(*******************************************************************************************************************)
//											Non operational system state
(*******************************************************************************************************************)
IF (gu8_SystemState = STANDBY_SYS OR gu8_SystemState = ERROR_SYS OR gu8_SystemState = OFF_SYS) THEN
	hq_BatteryDischargeMain_Rq			:=	FALSE;
	hq_Battery1ChargePrecharge_Rq		:=	FALSE;
	hq_Battery1ChargeMain_Rq			:=	FALSE;
	hq_Battery2ChargePrecharge_Rq		:=	FALSE;
	hq_BatteryDischargePrecharge_Rq		:=	FALSE;
	hq_Battery2ChargeMain_Rq			:=	FALSE;
	hton_Precharge_Timer				(IN := FALSE, PT := T#0MS);
	hton_PrechargeDisconnectBMS1_Timer	(IN := FALSE, PT := T#0MS);
	hton_PrechargeDisconnectBMS2_Timer	(IN := FALSE, PT := T#0MS);
	hton_Contactor_Delay				(IN := FALSE, PT := T#0MS);
	
(*******************************************************************************************************************)
//												System State Pre-Discharge
(*******************************************************************************************************************)
ELSIF (gu8_SystemState = DRIVE_SYS AND gr_BMS_BatteryVoltage > 0) THEN
	hr_MainConnectionVoltage	:=	gr_BMS_BatteryVoltage * PRECHARGEEND_VOLTAGE_PERC;
	hton_Contactor_Delay						(IN := TRUE, PT := T#500MS);
	IF (hton_Contactor_Delay.Q = TRUE) THEN
		IF ((gr_Sevcon1_DCLink_Voltage <= hr_MainConnectionVoltage OR
			 gr_Sevcon2_DCLink_Voltage <= hr_MainConnectionVoltage OR
			gu16_MCU_HighPowerVoltage <= hr_MainConnectionVoltage) AND
			DO_q_BatteryDischargeMain_DO = FALSE) THEN
			hq_BatteryDischargePrecharge_Rq	:=	TRUE;
			hton_PrechargeDisconnect_Timer		(IN := FALSE, PT := T#0MS);
			hton_MainContactorConnection_Delay	(IN := FALSE, PT := T#0MS);
(*******************************************************************************************************************)
//												System State Discharge
(*******************************************************************************************************************)			
		ELSIF ((gr_Sevcon1_DCLink_Voltage > hr_MainConnectionVoltage AND
				gr_Sevcon2_DCLink_Voltage > hr_MainConnectionVoltage AND
				gu16_MCU_HighPowerVoltage > hr_MainConnectionVoltage) OR
				DO_q_BatteryDischargeMain_DO = TRUE) THEN
			hton_MainContactorConnection_Delay(IN := TRUE, PT := T#100MS);
			IF (hton_MainContactorConnection_Delay.Q = TRUE) THEN
				hq_BatteryDischargeMain_Rq		:=	TRUE;
				hton_PrechargeDisconnect_Timer(IN := TRUE, PT := T#1S);
				IF (hton_PrechargeDisconnect_Timer.Q = TRUE) THEN
					hq_BatteryDischargePrecharge_Rq	:=	FALSE;
				END_IF
			END_IF
		ELSE
			hq_BatteryDischargeMain_Rq		:=	FALSE;
		END_IF
	END_IF
	hq_Battery1ChargePrecharge_Rq			:=	FALSE;
	hq_Battery1ChargeMain_Rq				:=	FALSE;
	hq_Battery2ChargePrecharge_Rq			:=	FALSE;
	hq_Battery2ChargeMain_Rq				:=	FALSE;
(*******************************************************************************************************************)
//												System State Charge
(******************************************************************************************************************)
ELSIF ((gu8_SystemState = PLUGIN_SYS AND
		Brusa1_Rx.S_ACDet = TRUE AND
		Brusa2_Rx.S_ACDet = TRUE AND
		gr_BMS_BatteryVoltage > 0)) THEN// Reset charge sequence if BMS safety drops out
		hton_Contactor_Delay(IN := DO_q_DrivetrainKL15C_DO, PT := T#500MS);
	IF (hton_Contactor_Delay.Q = TRUE) THEN
(*******************************************************************************************************************)
//												System State Pre-Charge Master
(******************************************************************************************************************)	
		IF OrionBMS1_RxConversion.Safety_OK THEN // Check that BMS1 safety is ok
			IF (Brusa1_RxConversion.DCHVVoltAct <= (gr_BMS1_Voltage * PRECHARGEEND_VOLTAGE_PERC) AND
				(DO_q_Battery1ChargeMain_DO = FALSE)) THEN
				hq_Battery1ChargePrecharge_Rq		  := TRUE;
(*******************************************************************************************************************)
//												System State Main-Charge Master
(******************************************************************************************************************)					
			ELSIF (Brusa1_RxConversion.DCHVVoltAct > (gr_BMS1_Voltage * PRECHARGEEND_VOLTAGE_PERC) OR
				DO_q_Battery1ChargeMain_DO) THEN
				hq_Battery1ChargeMain_Rq			  := TRUE;
				hton_PrechargeDisconnectBMS1_Timer(IN := TRUE, PT := T#1S);
				IF (hton_PrechargeDisconnectBMS1_Timer.Q) THEN
						hq_Battery1ChargePrecharge_Rq := FALSE;
				END_IF
			END_IF
		END_IF
(*******************************************************************************************************************)
//												System State Pre-Charge Slave
(******************************************************************************************************************)	
		IF OrionBMS2_RxConversion.Safety_OK THEN // Check that BMS2 safety is ok
			IF (Brusa2_RxConversion.DCHVVoltAct <= (gr_BMS2_Voltage * PRECHARGEEND_VOLTAGE_PERC) AND
				(DO_q_Battery2ChargeMain_DO = FALSE)) THEN
				hq_Battery2ChargePrecharge_Rq		  := TRUE;
(*******************************************************************************************************************)
//												System State Main-Charge Master
(******************************************************************************************************************)					
			ELSIF (Brusa2_RxConversion.DCHVVoltAct > (gr_BMS2_Voltage * PRECHARGEEND_VOLTAGE_PERC) OR
				DO_q_Battery2ChargeMain_DO) THEN
				hq_Battery2ChargeMain_Rq			  := TRUE;	
				hton_PrechargeDisconnectBMS2_Timer(IN := TRUE, PT := T#1S);
				IF (hton_PrechargeDisconnectBMS2_Timer.Q) THEN
					hq_Battery2ChargePrecharge_Rq	  := FALSE;
				END_IF
			END_IF
		END_IF
	ELSE
(*******************************************************************************************************************)
//												System Swich off all Contactor requests
(******************************************************************************************************************)			
		hq_Battery1ChargePrecharge_Rq		:=	FALSE;
		hq_Battery2ChargePrecharge_Rq		:=	FALSE;
		hq_Battery1ChargeMain_Rq			:=	FALSE;
		hq_Battery2ChargeMain_Rq			:=	FALSE;
	END_IF
	hq_BatteryDischargeMain_Rq				:=	FALSE;
	hq_BatteryDischargePrecharge_Rq			:=	FALSE;
ELSE
	hq_BatteryDischargeMain_Rq				:=	FALSE;
	hq_Battery1ChargePrecharge_Rq			:=	FALSE;
	hq_Battery1ChargeMain_Rq				:=	FALSE;
	hq_Battery2ChargePrecharge_Rq			:=	FALSE;
	hq_BatteryDischargePrecharge_Rq			:=	FALSE;
	hq_Battery2ChargeMain_Rq				:=	FALSE;
	hton_Precharge_Timer					(IN := FALSE, PT := T#0MS);
	hton_Contactor_Delay					(IN := FALSE, PT := T#0MS);
END_IF

(*******************************************************************************************************************)
//											Set the actual output values
// 		Current protection so if system current is over a certain value maintain contactor state to prevent welds
(******************************************************************************************************************)	
IF ((DOS_q_BatteryDischargeMain_DO <> hq_BatteryDischargeMain_Rq) AND
	(ABS(gs16_BMS_BatteryCurrent) > CONTACTORSWITCH_CURRENT_LIMIT)) THEN
	DO_q_BatteryDischargeMain_DO	:=	DOS_q_BatteryDischargeMain_DO;
ELSE
	DO_q_BatteryDischargeMain_DO	:=	hq_BatteryDischargeMain_Rq;
END_IF

IF ((DOS_q_Battery1ChargeMain_DO <> hq_Battery1ChargeMain_Rq) AND
	(ABS(gs16_BMS_BatteryCurrent) > CONTACTORSWITCH_CURRENT_LIMIT)) THEN
	DO_q_Battery1ChargeMain_DO	:=	DOS_q_Battery1ChargeMain_DO;
ELSE
	DO_q_Battery1ChargeMain_DO	:=	hq_Battery1ChargeMain_Rq;
END_IF

IF (DOS_q_Battery2ChargeMain_DO <> hq_Battery2ChargeMain_Rq AND
	(ABS(gs16_BMS_BatteryCurrent) > CONTACTORSWITCH_CURRENT_LIMIT)) THEN
	DO_q_Battery2ChargeMain_DO	:=	DOS_q_Battery2ChargeMain_DO;
ELSE
	DO_q_Battery2ChargeMain_DO	:=	hq_Battery2ChargeMain_Rq;
END_IF
(*******************************************************************************************************************)
//						Precharge contactors can change states to allow system connection								
(******************************************************************************************************************)		
DO_q_BatteryDischargePrecharge_DO	:=	hq_BatteryDischargePrecharge_Rq;
DO_q_Battery1ChargePrecharge_DO		:=	hq_Battery1ChargePrecharge_Rq;
DO_q_Battery2ChargePrecharge_DO		:=	hq_Battery2ChargePrecharge_Rq;

END_PROGRAM

// Application/UserCode/Brusa/Brusa2_Comms/Brusa2_RxConversion
PROGRAM Brusa2_RxConversion
VAR
ACVoltL1Act		:	UINT;
	ACVoltL2Act		:	UINT;
	ACVoltL3Act		:	UINT;
	ACCurrL1Act		:	SINT;
	ACCurrL2Act		:	SINT;
	ACCurrL3Act		:	SINT;
	ACPowTotAct		:	UINT;
	MaxTempAct		:	INT;
	TempCon			:	INT;
	DCHVAhAct			:	REAL;
	DCHVVoltAct			:	REAL;
	DCHVCurrAct			:	REAL;
	ACCurrMaxAct		:	REAL;
	ACCurrHWAvl			:	REAL;
	ACCurrMaxCP			:	REAL;
	TempCoolPlate		:	INT;		
END_VAR

ACVoltL1Act	:=	USINT_TO_UINT(Brusa2_Rx.ACVoltL1Act_Rx) * 2;
ACVoltL2Act	:=	USINT_TO_UINT(Brusa2_Rx.ACVoltL2Act_Rx) * 2;
ACVoltL3Act	:=	USINT_TO_UINT(Brusa2_Rx.ACVoltL3Act_Rx) * 2;
ACCurrL1Act	:=	USINT_TO_SINT(Brusa2_Rx.ACCurrL1Act_Rx) - 127;
ACCurrL2Act	:=	USINT_TO_SINT(Brusa2_Rx.ACCurrL2Act_Rx) - 127;
ACCurrL3Act	:=	USINT_TO_SINT(Brusa2_Rx.ACCurrL3Act_Rx) - 127;
ACPowTotAct	:=	USINT_TO_UINT(Brusa2_Rx.ACPowTotAct_Rx) * 100;
MaxTempAct	:=	USINT_TO_INT(Brusa2_Rx.MaxTempAct_Rx) - 50;
TempCon		:=	USINT_TO_INT(Brusa2_Rx.TempCon_Rx) - 50;
DCHVAhAct		:=	UINT_TO_REAL(Brusa2_Rx.DCHVAhAct_Rx) * 0.01;
DCHVVoltAct		:=	UINT_TO_REAL(Brusa2_Rx.DCHVVoltAct_Rx) * 0.1;
DCHVCurrAct		:=	UINT_TO_REAL(Brusa2_Rx.DCHVCurrAct_Rx) * 0.1 - 100;
ACCurrMaxAct	:=	UINT_TO_REAL(Brusa2_Rx.ACCurrMaxAct_Rx) * 0.1 -100;
ACCurrHWAvl		:=	USINT_TO_REAL(Brusa2_Rx.ACCurrHWAvl_Rx) * 0.5;
ACCurrMaxCP		:=	UINT_TO_REAL(Brusa2_Rx.ACCurrMaxCP_Rx) * 0.1;
TempCoolPlate	:=	USINT_TO_INT(Brusa2_Rx.TempCoolPlate_Rx) - 50;

END_PROGRAM

// Application/UserCode/Cooling Fan/Fan_Cooling
PROGRAM Fan_Cooling
VAR
	Cooling_Fan_MCU_SP				:	REAL	:=	30; // 30% requested
	Cooling_Fan_BRUSA_Charge_SP		:	REAL	:=	82;
	Cooling_Fan_BellP_Charge_SP		:	REAL	:=	82;	//	BellPower Charger 
	Cooling_Fan_DCDC_SP				:	REAL	:=	45; // Actual C Temp.
	Cooling_Fan_Request				:	BOOL	:=	FALSE;
	Cooling_Fan_DLY_Off				:	TOF;
	Run_On_Time						:	TIME	:=	T#60S;
END_VAR

(*****************************************************************************************************************)
//                       				   Radiator Cooling Fan
(*****************************************************************************************************************)

IF		((SUPPLY_Power1/100) > 25.0) AND	(NOT gq_EStop)				AND		// Do not run Fan if battery voltage is Low or EStopped
		(gr_MCU_ThermalIndicator		> Cooling_Fan_MCU_SP)			OR		// MCU
		(Brusa1_RxConversion.MaxTempAct	> Cooling_Fan_BRUSA_Charge_SP) 	OR		// BRUSA 1
		(Brusa2_RxConversion.MaxTempAct > Cooling_Fan_BRUSA_Charge_SP) 	OR		// BRUSA 2
	//	(BellPower_Charging				> Cooling_Fan_BellP_Charge_SP	OR		//	BellPower Charging	
		(BELDCDC_RxConversion.TempCoolant	> Cooling_Fan_DCDC_SP)		OR		// DCDC	
		HMI_Rx.PB_Cooling_Fan_Request									THEN	// Request from HMI
	
		Cooling_Fan_Request				:= TRUE;								// Fan Requested
ELSE
		Cooling_Fan_Request 			:= FALSE;								// Fan not Required
END_IF

		Cooling_Fan_DLY_Off		(IN := Cooling_Fan_Request, PT :=Run_On_Time);	// Fan run on time   (****provides hysteresis***)
IF 		(Cooling_Fan_DLY_Off.Q = TRUE) 									THEN
		DO_q_DrivetrainCoolingFan_DO	:=	TRUE;								// Fan Relay On
ELSE 
		DO_q_DrivetrainCoolingFan_DO	:=	FALSE;								// Fan Relay Off
END_IF

END_PROGRAM

// Application/UserCode/Cruise Control/CruiseControl
PROGRAM CruiseControl
VAR
	Cruise_Control_Button_DI: BOOL := FALSE;
	RS_CC: RS;
	CC_SetSpeed: REAL := 0;
	CC_Active: BOOL := FALSE;
	CC_VehicleSpeed: REAL := 0;
	SR_CC: SR;
	F_TRIG_CC_Set: F_TRIG;
	R_TRIG_CC_Set: R_TRIG;
	TESTSpeed: REAL := 0;
END_VAR

//Cruise Control

F_TRIG_CC_Set (CLK := DI_q_PB_Cruise_Control_DI);
R_TRIG_CC_Set (CLK := DI_q_PB_Cruise_Control_DI);

IF R_TRIG_CC_Set.Q AND gq_BrakeSwitch = FALSE AND (gu8_RegenSelector < 1) AND gu8_TractionLoss = 0 AND gu8_StabilityLoss = 0 THEN //LM added stab and trac event to cancel
	CC_Active := TRUE;
ELSIF CC_Active = TRUE THEN
	IF gq_BrakeSwitch = TRUE OR gu8_RegenSelector > 0 OR gu8_TractionLoss = 1 OR gu8_StabilityLoss = 1 THEN
	CC_Active := FALSE;
	END_IF
END_IF

IF CC_Active = TRUE THEN
	RS_CC (SET := DI_q_PB_Cruise_Control_DI = TRUE, RESET1 := F_TRIG_CC_Set.Q = TRUE);
END_IF

IF R_TRIG_CC_Set.Q = TRUE THEN
	SR_CC (SET1 := R_TRIG_CC_Set.Q = TRUE, RESET := (gq_BrakeSwitch = TRUE AND gu8_RegenSelector = 1));
END_IF

//IF SR_CC.Q1 = TRUE THEN
//	CC_SetSpeed := TESTSpeed;//gr_VehicleSpeed_kmph;
//END_IF

IF RS_CC.Q1 = TRUE THEN
	CC_SetSpeed := LIMIT (5, gr_VehicleSpeed_kmph, 57);//TESTSpeed;
END_IF

END_PROGRAM

// Application/UserCode/ePTO/ePTO_Control_1
PROGRAM ePTO_Control_1
VAR
	hu16_TORQUEREFHIGH	: UINT	:=	90; (*%*)
	hu16_TORQUEREFLOW	: UINT	:=	0;	(*%*)
	hu16_SPEEDTARGET	: UINT	:=	1150; (*RPM*)
	hs16_FAN_On_Temp	: INT	:=	60; (*degC*)
	hs16_FAN_Off_Temp	: INT	:=	50;	(*degC*)
	
	hton_CANOpen_Start_Timer	:	TON;
	hton_CANOpen_StartCommand_OtherAddress_Timer	:	TON;
	hu16_IdleSpeedTarget: UINT := 250;
	BinLiftTimer: TON;
	BinLiftTime: TIME := t#3s;
END_VAR


gu16_TrqHi	:=	(hu16_TORQUEREFHIGH * 50) + 5000;
gu16_TrqLo	:=	(hu16_TORQUEREFLOW * 50) + 5000;
gu8_Asym_Limits	:=	16#20;

IF ((gs16_InverterTemp > hs16_FAN_On_Temp) OR (gs16_MotorTemp > hs16_FAN_On_Temp)) THEN
	gu8_DIGITAL1	:=	16#80;
ELSIF ((gs16_InverterTemp < hs16_FAN_Off_Temp) AND (gs16_MotorTemp < hs16_FAN_Off_Temp)) THEN
	gu8_DIGITAL1	:=	16#0;
END_IF

BinLiftTimer (IN:= (gq_Gear_Drive = TRUE OR gq_Gear_Reverse = TRUE), PT:= BinLiftTime);

IF (DOS_q_BatteryDischargeMain_DO = TRUE) THEN
	(*Activate Motor*)
	IF (gu8_ePTO_ActivationByte <> 0) OR (BinLiftTimer.Q = FALSE AND gq_Gear_Neutral = FALSE) THEN
		gu16_Skai_SpeedTarget	:=	hu16_SPEEDTARGET + 32768;
		gq_ePTO_Activate	:=	TRUE;
	ELSE
		gu16_Skai_SpeedTarget	:=	hu16_IdleSpeedTarget + 32768; (*added to allow permanent running of ePTO*)
		gq_ePTO_Activate	:=	TRUE(*FALSE*);
	END_IF
ELSE
	gu16_Skai_SpeedTarget	:=	32768; (*Offset so value is actually 0*)
	gq_ePTO_Activate	:=	FALSE;
END_IF


(*CANOpen*)
hton_CANOpen_Start_Timer(IN := TRUE, PT := T#5S);
hton_CANOpen_StartCommand_OtherAddress_Timer(IN := hton_CANOpen_Start_Timer.Q, PT := T#1S);
IF (hton_CANOpen_Start_Timer.Q = TRUE) THEN
	gu8_CANOpen_Command	:=	16#01;
	gu8_CANOpen_NodeAddress	:=	16#7A;
ELSIF (hton_CANOpen_StartCommand_OtherAddress_Timer.Q = TRUE) THEN
	gu8_CANOpen_Command	:=	16#01;
	gu8_CANOpen_NodeAddress	:=	16#7B;
ELSE
	gu8_CANOpen_Command	:=	16#81;
	gu8_CANOpen_NodeAddress	:=	16#7A;
END_IF

DO_q_ePTO_Fan_DO	:=	gq_ePTO_Activate;

END_PROGRAM

// Application/UserCode/ePTO/EPTO_Rx_1
PROGRAM EPTO_Rx_1
VAR
	ePTO_Rx			:	Receive_CAN4_STD;
	ePTO_Dennis_Rx	:	Receive_CAN4_EXD;
	SkaiUnit_Temp_Rx	:	Receive_CAN4_STD;
END_VAR


ePTO_Rx		(u32_COBID	:=	16#141,
						q_NewData => ,
						au8_Data => ,
						u8_Length => 		);
						
ePTO_Dennis_Rx (u32_COBID	:=	16#2CFF1355,
						q_NewData => ,
						au8_Data => ,
						u8_Length => 		);
						
SkaiUnit_Temp_Rx (u32_COBID	:=	16#1BA,
						q_NewData => ,
						au8_Data => ,
						u8_Length => 		);

IF (gu8_ChassisType = CHASSIS_DENNIS) THEN
	gu8_ePTO_ActivationByte	:=	ePTO_Dennis_Rx.au8_Data[3]; (*4*)
ELSE
	gu8_ePTO_ActivationByte	:=	ePTO_Rx.au8_Data[4];				
END_IF					

gs16_InverterTemp	:= SkaiUnit_Temp_Rx.au8_Data[0] - 40;
gs16_MotorTemp		:= SkaiUnit_Temp_Rx.au8_Data[1] - 40; (*Use this for the ePTO activation instead of the boolean trigger*)

END_PROGRAM

// Application/UserCode/ePTO/EPTO_Tx_1
PROGRAM EPTO_Tx_1
VAR
	MercCurrentGear1_Tx	:	EPEC_CANVXD.Msg;
	MercLHFWheelSpd_Tx	:	EPEC_CANVXD.Msg;
	MercCurrentGear2_Tx	:	EPEC_CANVXD.Msg;
	MercControlRPM_Tx	:	EPEC_CANVXD.Msg;
	ePTO_OilRq_Tx		:	EPEC_CANVXD.Msg;
	ePTO_Speed_47A_Tx	:	EPEC_CANVXD.Msg;
	ePTO_Torque_57A_Tx	:	EPEC_CANVXD.Msg;
	ePTO_NMT_Tx			:	EPEC_CANVXD.Msg;
	
	
	hton_MercePTO_TxTimer	:	TON;
END_VAR


{region "Data Allocation"}
(*Merc*)
MercCurrentGear1_Tx.ID := 16#18FE61EB OR EPEC_CANVXD.MASK_29BIT;
MercCurrentGear1_Tx.Data[0]	:=	0;
MercCurrentGear1_Tx.Data[1]	:=	gu8_CurrentGear2;
MercCurrentGear1_Tx.Data[2]	:=	0;
MercCurrentGear1_Tx.Data[3]	:=	0;
MercCurrentGear1_Tx.Data[4]	:=	0;
MercCurrentGear1_Tx.Data[5]	:=	0;
MercCurrentGear1_Tx.Data[6]	:=	0;
MercCurrentGear1_Tx.Data[7]	:=	0;
MercCurrentGear1_Tx.Len		:=	8;

MercLHFWheelSpd_Tx.ID := 16#0CFE5FEB OR EPEC_CANVXD.MASK_29BIT;
MercLHFWheelSpd_Tx.Data[0]	:=	0;
MercLHFWheelSpd_Tx.Data[1]	:=	0;
MercLHFWheelSpd_Tx.Data[2]	:=	0;
MercLHFWheelSpd_Tx.Data[3]	:=	03;
MercLHFWheelSpd_Tx.Data[4]	:=	20;
MercLHFWheelSpd_Tx.Data[5]	:=	0;
MercLHFWheelSpd_Tx.Data[6]	:=	UINT_TO_USINT(gu16_Bob_LeftFront_CAN);
MercLHFWheelSpd_Tx.Data[7]	:=	UINT_TO_USINT(SHR(gu16_Bob_LeftFront_CAN, 8));
MercLHFWheelSpd_Tx.Len		:=	8;

MercCurrentGear2_Tx.ID := 16#14FE80EB OR EPEC_CANVXD.MASK_29BIT;
MercCurrentGear2_Tx.Data[0]	:=	0;
MercCurrentGear2_Tx.Data[1]	:=	gu8_CurrentGear2;
MercCurrentGear2_Tx.Data[2]	:=	0;
MercCurrentGear2_Tx.Data[3]	:=	0;
MercCurrentGear2_Tx.Data[4]	:=	0;
MercCurrentGear2_Tx.Data[5]	:=	0;
MercCurrentGear2_Tx.Data[6]	:=	0;
MercCurrentGear2_Tx.Data[7]	:=	0;
MercCurrentGear2_Tx.Len		:=	8;

MercControlRPM_Tx.ID := 16#0CFE62C9 OR EPEC_CANVXD.MASK_29BIT;
MercControlRPM_Tx.Data[0]	:=	0;
MercControlRPM_Tx.Data[1]	:=	0;
MercControlRPM_Tx.Data[2]	:=	0;
MercControlRPM_Tx.Data[3]	:=	16#FA;
MercControlRPM_Tx.Data[4]	:=	0;
MercControlRPM_Tx.Data[5]	:=	0;
MercControlRPM_Tx.Data[6]	:=	0;
MercControlRPM_Tx.Data[7]	:=	0;
MercControlRPM_Tx.Len		:=	8;
	 
ePTO_OilRq_Tx.ID			:=	16#0CFF1355 OR EPEC_CANVXD.MASK_29BIT;
ePTO_OilRq_Tx.Data[0]		:=	0;
ePTO_OilRq_Tx.Data[1]		:=	0;
ePTO_OilRq_Tx.Data[2]		:=	0;
ePTO_OilRq_Tx.Data[3]		:=	0;
ePTO_OilRq_Tx.Data[3].0		:=	gq_ePTO_Activate;
ePTO_OilRq_Tx.Data[4]		:=	0;
ePTO_OilRq_Tx.Data[5]		:=	0;
ePTO_OilRq_Tx.Data[6]		:=	0;
ePTO_OilRq_Tx.Data[7]		:=	0;
ePTO_OilRq_Tx.Len			:=	8;
(**)


ePTO_Speed_47A_Tx.ID		:=	16#47A;
ePTO_Speed_47A_Tx.Data[0]	:=	UINT_TO_USINT(gu16_TrqHi);
ePTO_Speed_47A_Tx.Data[1]	:=	UINT_TO_USINT(SHR(gu16_TrqHi, 8));
ePTO_Speed_47A_Tx.Data[2]	:=	UINT_TO_USINT(gu16_Skai_SpeedTarget);
ePTO_Speed_47A_Tx.Data[3]	:=	UINT_TO_USINT(SHR(gu16_Skai_SpeedTarget, 8));
ePTO_Speed_47A_Tx.Data[4]	:=	(BOOL_TO_USINT(gq_ePTO_Activate) * 2);
ePTO_Speed_47A_Tx.Data[5]	:=	gu8_Asym_Limits + gu8_DIGITAL1;
ePTO_Speed_47A_Tx.Data[6]	:=	0;
ePTO_Speed_47A_Tx.Data[7]	:=	0;
ePTO_Speed_47A_Tx.Len		:=	8;
	 
ePTO_Torque_57A_Tx.ID		:=	16#57A;
ePTO_Torque_57A_Tx.Data[0]	:=	UINT_TO_USINT(gu16_TrqHi);
ePTO_Torque_57A_Tx.Data[1]	:=	UINT_TO_USINT(SHR(gu16_TrqHi, 8));
ePTO_Torque_57A_Tx.Data[2]	:=	UINT_TO_USINT(gu16_TrqLo);
ePTO_Torque_57A_Tx.Data[3]	:=	UINT_TO_USINT(SHR(gu16_TrqLo, 8));
ePTO_Torque_57A_Tx.Data[4]	:=	0;
ePTO_Torque_57A_Tx.Data[5]	:=	0;
ePTO_Torque_57A_Tx.Data[6]	:=	0;
ePTO_Torque_57A_Tx.Data[7]	:=	0;
ePTO_Torque_57A_Tx.Len		:=	8;

(*CANOpen*)
ePTO_NMT_Tx.ID				:=	16#00;
ePTO_NMT_Tx.Data[0]			:=	gu8_CANOpen_Command;
ePTO_NMT_Tx.Data[1]			:=	gu8_CANOpen_NodeAddress;
ePTO_NMT_Tx.Len				:=	8;
{endregion}

	 
(**************************************************************************************************************************************************)
{region "Send Messages"}
(*Transmit*)
hton_MercePTO_TxTimer(IN := NOT(hton_MercePTO_TxTimer.Q), PT := T#100MS);
IF (hton_MercePTO_TxTimer.Q = TRUE) THEN
	IF (gu8_ChassisType = CHASSIS_BOB OR gu8_ChassisType = CHASSIS_ESTARGLIDER) THEN
		G_CAN4_Channel.SendMessage(i_pMSG:=ADR(MercCurrentGear1_Tx)); 
		G_CAN4_Channel.SendMessage(i_pMSG:=ADR(MercLHFWheelSpd_Tx)); 
		G_CAN4_Channel.SendMessage(i_pMSG:=ADR(MercCurrentGear2_Tx)); 
		G_CAN4_Channel.SendMessage(i_pMSG:=ADR(MercControlRPM_Tx));
	ELSIF (gu8_ChassisType = CHASSIS_DENNIS) THEN
		;
	END_IF
 
	G_CAN4_Channel.SendMessage(i_pMSG:=ADR(ePTO_Speed_47A_Tx));
	G_CAN4_Channel.SendMessage(i_pMSG:=ADR(ePTO_Torque_57A_Tx)); 
	G_CAN4_Channel.SendMessage(i_pMSG:=ADR(ePTO_OilRq_Tx)); 
		 
	G_CAN4_Channel.SendMessage(i_pMSG:=ADR(ePTO_NMT_Tx)); 
END_IF

{end_region}

END_PROGRAM

// Application/UserCode/Fault Handler/FaultDetection_1
PROGRAM FaultDetection_1
VAR
	hq_Dennis_CommsErr			:	BOOL;
	gq_BMS1_Orion_Error			:	BOOL;
	gq_BMS2_Orion_Error			:	BOOL;
	gq_BMS1_Error				:	BOOL;
	gq_BMS2_Error				:	BOOL;
	gq_BMS_Error				:	BOOL;
	gq_DCDC_Bel_Error			:	BOOL;
	gq_MCU_Error				:	BOOL;
	gq_NLG1_Error				:	BOOL;
	gq_NLG2_Error				:	BOOL;
	gq_Sevcon_Steer_Error		:	BOOL;
	gq_Sevcon_Compressor_Error	:	BOOL;
	gq_LV_Error					:	BOOL;// 24V Batteries too Low Error
END_VAR
VAR CONSTANT
	FAULTOFF_STAT				:	USINT	:=	13;
	Low_24V_Battery_Voltage_SP	:	USINT	:=	21;
END_VAR

(**********************************************************************************)
//									Faults & Errors
(**********************************************************************************)

(**********************************************************************************)
// 									Orion BMS1 Faults
(**********************************************************************************)

IF (gu8_BMSType = BMS_ORION) THEN
	IF(	//OrionBMS1_DTCFlag1_0A07_DischargeLimitEnforcementFault= TRUE OR
		OrionBMS1_DTCFlag1_0A08_ChargerSafetyRelayFault			= TRUE OR
		OrionBMS1_DTCFlag1_0A09_InternalHardwareFault			= TRUE OR
		OrionBMS1_DTCFlag1_0A0A_InternalHeatskinkThermistorFault= TRUE OR
		OrionBMS1_DTCFlag1_0A0B_InternalSoftwareFault			= TRUE OR
		OrionBMS1_DTCFlag1_0A0C_HighestCellVoltageTooHighFault	= TRUE OR 
		OrionBMS1_DTCFlag1_0A0E_LowestCellVoltageTooLowFault	= TRUE OR	
		OrionBMS1_DTCFlag1_0A10_PackTooHotFault					= TRUE OR	
		(*DTC2 Flags*)
		OrionBMS1_DTCFlags2_0A1F_InternalCommunicationFault		= TRUE OR	
		//OrionBMS1_DTCFlags2_0A12_CellBalancingStruckOffFault	= TRUE OR	
		//OrionBMS1_DTCFlags2_0A80_WeakCellFault				= TRUE OR*)
		OrionBMS1_DTCFlags2_0AFA_LowCellVoltageFault			= TRUE OR			
		OrionBMS1_DTCFlags2_0A04_OpenWiringFault				= TRUE OR
		OrionBMS1_DTCFlags2_0AC0_CurrentSensorFault				= TRUE OR				
		OrionBMS1_DTCFlags2_0A0D_HighestCellVoltageOver5vFault	= TRUE OR		
		OrionBMS1_DTCFlags2_0A0F_CellASICFault					= TRUE OR
		OrionBMS1_DTCFlags2_0A02_WeakPackFault					= TRUE OR				
		//OrionBMS1_DTCFlags2_0A81_FanMonitorFault				= TRUE OR				
		//OrionBMS1_DTCFlags2_0A9C_ThermistorFault				= TRUE OR			
		OrionBMS1_DTCFlags2_0100_ExternalCommunicationFault		= TRUE OR		
		OrionBMS1_DTCFlags2_0560_RedundantPowerSupplyFault		= TRUE OR	
		OrionBMS1_DTCFlags2_0AA6_HighVoltageIsolatonFault		= TRUE OR
		OrionBMS1_DTCFlags2_0A05_InputPowerSupplyFault			= TRUE OR	
		//OrionBMS1_DTCFlags2_0A06_ChargeLimitEnforcementFault	= TRUE OR
		gq_OrionBMS1_CommsLoss 									= TRUE) THEN
			gq_BMS1_Orion_Error									:=	TRUE;
	ELSE
			gq_BMS1_Orion_Error									:=	FALSE;
	END_IF

(**********************************************************************************)	
// 									Orion BMS2 Faults	
(**********************************************************************************)

	IF(//OrionBMS2_DTCFlag1_0A07_DischargeLimitEnforcementFault= TRUE OR
		OrionBMS2_DTCFlag1_0A08_ChargerSafetyRelayFault			= TRUE OR
		OrionBMS2_DTCFlag1_0A09_InternalHardwareFault			= TRUE OR
		OrionBMS2_DTCFlag1_0A0A_InternalHeatskinkThermistorFault= TRUE OR
		OrionBMS2_DTCFlag1_0A0B_InternalSoftwareFault			= TRUE OR
		OrionBMS2_DTCFlag1_0A0C_HighestCellVoltageTooHighFault	= TRUE OR 
		OrionBMS2_DTCFlag1_0A0E_LowestCellVoltageTooLowFault	= TRUE OR	
		OrionBMS2_DTCFlag1_0A10_PackTooHotFault					= TRUE OR	
		(*DTC2 Flags*)
		OrionBMS2_DTCFlags2_0A1F_InternalCommunicationFault		= TRUE OR	
		//OrionBMS2_DTCFlags2_0A12_CellBalancingStruckOffFault	= TRUE OR	
		//OrionBMS2_DTCFlags2_0A80_WeakCellFault				= TRUE OR
		OrionBMS2_DTCFlags2_0AFA_LowCellVoltageFault			= TRUE OR			
		OrionBMS2_DTCFlags2_0A04_OpenWiringFault				= TRUE OR
		OrionBMS2_DTCFlags2_0AC0_CurrentSensorFault				= TRUE OR				
		OrionBMS2_DTCFlags2_0A0D_HighestCellVoltageOver5vFault	= TRUE OR		
		OrionBMS2_DTCFlags2_0A0F_CellASICFault					= TRUE OR
		OrionBMS2_DTCFlags2_0A02_WeakPackFault					= TRUE OR				
		//OrionBMS2_DTCFlags2_0A81_FanMonitorFault				= TRUE OR				
		//OrionBMS2_DTCFlags2_0A9C_ThermistorFault				= TRUE OR			
		OrionBMS2_DTCFlags2_0100_ExternalCommunicationFault		= TRUE OR		
		OrionBMS2_DTCFlags2_0560_RedundantPowerSupplyFault		= TRUE OR	
		OrionBMS2_DTCFlags2_0AA6_HighVoltageIsolatonFault		= TRUE OR
		OrionBMS2_DTCFlags2_0A05_InputPowerSupplyFault			= TRUE OR	
		//OrionBMS2_DTCFlags2_0A06_ChargeLimitEnforcementFault	= TRUE OR
		gq_OrionBMS2_CommsLoss 									= TRUE) THEN
			gq_BMS2_Orion_Error									:=	TRUE;
	ELSE
			gq_BMS2_Orion_Error									:=	FALSE;
	END_IF
END_IF

(**********************************************************************************)
// 									Orion BMS Faults
(**********************************************************************************)
	 
IF (gq_BMS1_Orion_Error = TRUE) THEN
	gq_BMS1_Error	:=	TRUE;
ELSE
	gq_BMS1_Error	:=	FALSE;		 
END_IF

IF (gq_BMS2_Orion_Error = TRUE) THEN
	gq_BMS2_Error	:=	TRUE;
ELSE 
	gq_BMS2_Error	:=	FALSE;
END_IF

IF (gq_BMS1_Error = TRUE OR gq_BMS2_Error = TRUE) THEN
	gq_BMS_Error	:=	TRUE;
ELSE
	gq_BMS_Error	:=	FALSE;
END_IF

(**********************************************************************************)
// 									BelPower DCDC Faults
(**********************************************************************************)

IF (BELDCDC_Rx.Fault_InputUV 					= TRUE OR
	BELDCDC_Rx.Fault_InputOV 					= TRUE OR
	(*BELDCDC_Rx.gq_BelDCDC_flt_OutputUV		= TRUE OR*)
	BELDCDC_Rx.Fault_OutputOV 					= TRUE OR
	(*BELDCDC_Rx.gq_BelDCDC_flt_OutputOC 		= TRUE OR*) (*Need to reenable this when possible*)
	BELDCDC_Rx.Fault_OTP 						= TRUE OR
	BELDCDC_Rx.Fault_I2CFault 					= TRUE OR
	BELDCDC_Rx.Fault_CANFault 					= TRUE OR
	BELDCDC_Rx.Fault_EEPROM_CRCFault 			= TRUE OR
	BELDCDC_Rx.Fault_ShortCircuit 				= TRUE OR
	BELDCDC_Rx.Fault_ThermistorFault 			= TRUE OR
	BELDCDC_Rx.Fault_Overload 					= TRUE OR
	BELDCDC_Rx.Fault_OutputOVLatch 				= TRUE OR
	BELDCDC_Rx.Fault_ReversePolarity 			= TRUE OR
	BELDCDC_Rx.Warning_CoolantOTP 				= TRUE OR
	BELDCDC_Rx.Warning_CurrentLimiting 			= TRUE OR
	BELDCDC_Rx.CommsLoss)							THEN
	gq_DCDC_Bel_Error							:=	TRUE;
ELSE
	gq_DCDC_Bel_Error							:=	FALSE;
END_IF

(**********************************************************************************)
// 									MCU  Faults
(**********************************************************************************)

IF (gq_MCU_Fault_PhaseToChassis 		= TRUE OR
	gq_MCU_Fault_InterlockBatteryCable 	= TRUE OR
	gq_MCU_Fault_InterlockMotorCable 	= TRUE OR
	gq_MCU_Fault_DriveCoverWasOpened 	= TRUE OR
	gq_MCU_Fault_PhaseToChassisStatus 	= TRUE OR
	(gq_MCU_CommsLoss = TRUE AND gu8_SystemState = DRIVE_SYS)) THEN
	gq_MCU_Error	:=	TRUE;
ELSE
	gq_MCU_Error	:=	FALSE;
END_IF

(**********************************************************************************)
// 									BRUSA1 Faults
(**********************************************************************************)

IF (gu8_ChargerType = CHARGER_BRUSA) THEN
	IF (Brusa1_Rx.E_WrongHW 		= TRUE OR
		Brusa1_Rx.E_WrongFPGA 		= TRUE OR
		Brusa1_Rx.E_EPGAInit 		= TRUE OR
		Brusa1_Rx.E_NVSRam 			= TRUE OR
		Brusa1_Rx.E_Flash 			= TRUE OR
		Brusa1_Rx.E_OSTrap 			= TRUE OR
		Brusa1_Rx.E_HVIsoPos 		= TRUE OR
		Brusa1_Rx.E_HVIsoNeg 		= TRUE OR
		Brusa1_Rx.E_Internal 		= TRUE OR
		Brusa1_Rx.E_TempInt 		= TRUE OR
		Brusa1_Rx.E_DCHVVoltRed 	= TRUE OR
		Brusa1_Rx.E_IntSupply 		= TRUE OR
		Brusa1_Rx.E_CANMsgLost 		= TRUE OR
		Brusa1_Rx.E_CANValue 		= TRUE OR
		Brusa1_Rx.E_ACInterruption 	= TRUE OR
		Brusa1_Rx.E_DCHVVoltRange 	= TRUE OR
		Brusa1_Rx.E_TempCon 		= TRUE OR
		Brusa1_Rx.E_ConLocked 		= TRUE OR
		Brusa1_Rx.E_Interlock 		= TRUE OR
		Brusa1_Rx.E_Crash 			= TRUE OR
		Brusa1_Rx.E_PRELOAD 		= TRUE OR
		Brusa1_Rx.E_BURST 			= TRUE OR
		Brusa1_Rx.E_TPON 			= TRUE OR
		Brusa1_Rx.E_UZK 			= TRUE OR
		Brusa1_Rx.E_LatchFPGA 		= TRUE OR
		Brusa1_Rx.E_OverTemp 		= TRUE OR
		Brusa1_Rx.CommsLoss = TRUE)	 THEN
		gq_NLG1_Error	:=	TRUE;
	ELSE
		gq_NLG1_Error	:=	FALSE;
	END_IF

(**********************************************************************************)	
// 									BRUSA2 Faults
(**********************************************************************************)
			  
	IF (Brusa2_Rx.E_WrongHW 		= TRUE OR
		Brusa2_Rx.E_WrongFPGA 		= TRUE OR
		Brusa2_Rx.E_EPGAInit		= TRUE OR
		Brusa2_Rx.E_NVSRam 			= TRUE OR
		Brusa2_Rx.E_Flash 			= TRUE OR
		Brusa2_Rx.E_OSTrap 			= TRUE OR
		Brusa2_Rx.E_HVIsoPos 		= TRUE OR
		Brusa2_Rx.E_HVIsoNeg 		= TRUE OR
		Brusa2_Rx.E_Internal		= TRUE OR
		Brusa2_Rx.E_TempInt 		= TRUE OR
		Brusa2_Rx.E_DCHVVoltRed 	= TRUE OR
		Brusa2_Rx.E_IntSupply		= TRUE OR
		Brusa2_Rx.E_CANMsgLost		= TRUE OR
		Brusa2_Rx.E_CANValue		= TRUE OR
		Brusa2_Rx.E_ACInterruption = TRUE OR
		Brusa2_Rx.E_DCHVVoltRange 	= TRUE OR
		Brusa2_Rx.E_TempCon			= TRUE OR
		Brusa2_Rx.E_ConLocked 		= TRUE OR
		Brusa2_Rx.E_Interlock 		= TRUE OR
		Brusa2_Rx.E_Crash 			= TRUE OR
		Brusa2_Rx.E_PRELOAD 		= TRUE OR
		Brusa2_Rx.E_BURST 			= TRUE OR
		Brusa2_Rx.E_TPON 			= TRUE OR
	    Brusa2_Rx.E_UZK 			= TRUE OR
		Brusa2_Rx.E_LatchFPGA 		= TRUE OR
		Brusa2_Rx.E_OverTemp 		= TRUE OR
		Brusa2_Rx.CommsLoss 		= TRUE) THEN
		gq_NLG2_Error				:=	TRUE;
	ELSE
			gq_NLG2_Error			:=	FALSE;
	END_IF 
	
END_IF

(**********************************************************************************)
// 									Sevcon Faults
(**********************************************************************************)

IF (gu8_Sevcon1_InverterStatus = FAULTOFF_STAT OR
	(gq_Sevcon1_CommsLoss = TRUE AND gu8_SystemState = DRIVE_SYS)) THEN
	gq_Sevcon_Steer_Error	:=	TRUE;
ELSE
	gq_Sevcon_Steer_Error	:=	FALSE;
END_IF

IF (gu8_Sevcon2_InverterStatus = FAULTOFF_STAT OR
	(gq_Sevcon2_CommsLoss = TRUE AND gu8_SystemState = DRIVE_SYS)) THEN
	gq_Sevcon_Compressor_Error	:=	TRUE;
ELSE
	gq_Sevcon_Compressor_Error	:=	FALSE;
END_IF

(**********************************************************************************)
// 									24VDC Faults
(**********************************************************************************)

IF ((SUPPLY_Power1/100) < Low_24V_Battery_Voltage_SP)  THEN (*SUPPLY_Power1*)
	gq_LV_Error	:=	TRUE;
ELSE
	gq_LV_Error	:=	FALSE; 
END_IF

(**********************************************************************************)
// 									eCompact Faults
(**********************************************************************************)

 IF ((gq_Dennis_CAN1_CommsLoss = TRUE OR CAN4_Rx.Handbrake_Rx_Timer.Q = TRUE) AND
	  gu8_ChassisType = CHASSIS_DENNIS AND gu8_SystemState = DRIVE_SYS) THEN
	hq_Dennis_CommsErr	:=	TRUE;
 ELSE
	hq_Dennis_CommsErr	:=	FALSE;	  
 END_IF

 (**********************************************************************************)
 // 									Global Faults
(**********************************************************************************)
	 
IF (gq_BMS_Error				OR
	gq_DCDC_Bel_Error			OR
	gq_MCU_Error				OR
	Brusa1_Rx.S_Err				OR					//***************************************WRONG!!!!!!!!!!!!!!!!!!!!!!!!!!!
	gq_NLG2_Error				OR
	gq_Sevcon_Steer_Error		OR
	gq_Sevcon_Compressor_Error	OR
	gq_LV_Error					OR
	hq_Dennis_CommsErr			OR
	gq_EStop)	 			 THEN
		gq_SystemError	:=	TRUE;
ELSE
		gq_SystemError	:=	FALSE;
END_IF

END_PROGRAM

// Application/UserCode/Functions/Update_1
(*==============================================================================================================*)
(*     Function to handle state updates                                                                         *)
(*==============================================================================================================*)
FUNCTION Update_1 : BOOL
VAR_INPUT
 ptUp        : POINTER TO tUpdate; // Pointer to screen update

END_VAR
VAR
END_VAR

(*==============================================================================================================*)
(*     Function to handle state updates                                                                         *)
(*==============================================================================================================*)
IF (ptUp^.Next <> ptUp^.Step) THEN                         // New State Requested?	
	ptUp^.Last			:= ptUp^.Step;                     // Save Current State
	ptUp^.Step			:= ptUp^.Next;                     // Set New State
	ptUp^.Seq  			:= (ptUp^.Seq * 256) + ptUp^.Next; // Shift In New State
	ptUp^.Tmr			:= 0;                              // Reset State Timer
ELSIF (ptUp^.Tmr <> 65535) THEN                            // Timer Less than max?
	ptUp^.Tmr			:= (ptUp^.Tmr + 1);                // Increment Timer
END_IF

END_FUNCTION

// Application/UserCode/Heater/Heater_Control_1
PROGRAM Heater_Control_1
VAR
	PWR_2kW				:	BYTE	:=	20;
	PWR_4kW				:	BYTE	:=	40;
	PWR_8kW				:	BYTE	:=	80;
	HEATER_TEMP_60C		:	BYTE 	:= 110;// Temperature request 110(dec) - 50 deg C = 60degC
	HEATER_TEMP_50C		:	BYTE 	:= 100;// Temperature request 100(dec) - 50 deg C = 50degC
	HEATER_TEMP_40C		:	BYTE 	:= 90; // Temperature request 90(dec) - 50 deg C = 40degC
	Heater_Enable		:	BOOL 	:= FALSE;
	Heater_PWR			:	BYTE	:= 0;
	Heater_Temperature	: 	BYTE 	:= 0;
	Heater_Pump_Rq		:	BOOL 	:= FALSE; // Pump Relay Required
END_VAR

(*****************************************************************************************************)
//									Cabin Heater Control
(*****************************************************************************************************)

IF		HMI_Rx.Heater_Enable AND DO_q_BatteryDischargeMain_DO AND
		DI_q_VehicleKL15_DI AND (NOT gq_EStop) THEN  // Need to add DCL here
		Heater_Pump_Rq			:=	TRUE;
		Heater_Enable			:=	TRUE;
ELSE
		Heater_PWR				:=	0;
		Heater_Temperature		:=	0;
		Heater_Pump_Rq			:=	FALSE;
		Heater_Enable			:=	FALSE;
END_IF

IF 		(Heater_Pump_Rq = TRUE) AND (HMI_Rx.Heater_Low = TRUE) THEN
		Heater_PWR				:=	PWR_8kW;
		Heater_Temperature		:=	HEATER_TEMP_40C;
ELSIF 	(Heater_Pump_Rq = TRUE) AND (HMI_Rx.Heater_Med = TRUE) THEN
		Heater_PWR				:=	PWR_8kW;
		Heater_Temperature		:=	HEATER_TEMP_50C; 
ELSIF 	(Heater_Pump_Rq = TRUE) AND (HMI_Rx.Heater_Hi = TRUE) THEN
		Heater_PWR				:=	PWR_8kW;
		Heater_Temperature		:=	HEATER_TEMP_60C;
END_IF

IF (NOT DO_q_BatteryDischargeMain_DO) OR (NOT DI_q_VehicleKL15_DI) THEN
		Heater_PWR				:=	0;
		Heater_Temperature		:=	0;
		Heater_Pump_Rq			:=	FALSE;
		Heater_Enable			:=	FALSE;
END_IF

		DO_q_HeaterOut_DI		:=	Heater_Pump_Rq;

END_PROGRAM

// Application/UserCode/Heater/Heater_Rx_1
PROGRAM Heater_Rx_1
VAR
END_VAR

//Awaiting all the Data From the heater LDF
// All taken care of in HMI Code.
//So there MF>

END_PROGRAM

// Application/UserCode/Heater/Heater_Tx_1
PROGRAM Heater_Tx_1
VAR
	ht_CAN4_Heater_Tx		:	EPEC_CANVXD.Msg;
	ht_CAN4_OldHeater_Tx	:	EPEC_CANVXD.Msg;
	
END_VAR

//r2
ht_CAN4_Heater_Tx.ID			:=	16#023;
ht_CAN4_Heater_Tx.Data[0]		:=	Heater_Control.Heater_PWR;
ht_CAN4_Heater_Tx.Data[1]		:=	Heater_Control.Heater_Temperature;
ht_CAN4_Heater_Tx.Data[2]		:=	0;
ht_CAN4_Heater_Tx.Data[3].3		:=	Heater_Control.Heater_Enable;
ht_CAN4_Heater_Tx.Data[4]		:=	0;
ht_CAN4_Heater_Tx.Data[5]		:=	0;
ht_CAN4_Heater_Tx.Data[6]		:=	0;
ht_CAN4_Heater_Tx.Data[7]		:=	0;
ht_CAN4_Heater_Tx.Len			:=	8;

ht_CAN4_OldHeater_Tx.ID			:=	16#066;
ht_CAN4_OldHeater_Tx.Data[0].0	:=	Heater_Control.Heater_Enable;
ht_CAN4_OldHeater_Tx.Data[1]	:=	Heater_Control.Heater_PWR;
ht_CAN4_OldHeater_Tx.Data[2]	:=	0;
ht_CAN4_OldHeater_Tx.Data[3]	:=	0;
ht_CAN4_OldHeater_Tx.Data[4]	:=	0;
ht_CAN4_OldHeater_Tx.Data[5]	:=	0;
ht_CAN4_OldHeater_Tx.Data[6]	:=	0;
ht_CAN4_OldHeater_Tx.Data[7]	:=	0;
ht_CAN4_OldHeater_Tx.Len		:=	8;

G_CAN4_Channel.SendMessage(i_pMSG:=ADR(ht_CAN4_Heater_Tx));
G_CAN4_Channel.SendMessage(i_pMSG:=ADR(ht_CAN4_OldHeater_Tx));

END_PROGRAM

// Application/UserCode/HMI/HMI_Rx_1
PROGRAM HMI_Rx_1
VAR
	HMI_Commands_Rx		:	Receive_CAN4_STD;
	
	EStop_Bad                   :	BOOL;
	Hand_Brake_On				:	BOOL;	
	Heater_Enable				:	BOOL;
	StopChargeRq             	:	BOOL;   // Stop charge request from HMI
	Heater_Low					:	BOOL;
	Heater_Med					:	BOOL;
	Heater_Hi					:	BOOL;
	SW_Isolation_On				:	BOOL;	// Isolation Switch On For CATL Only.
	
	PB_BMS1_DTC_Reset			:	BOOL;
	PB_BMS2_DTC_Reset			:	BOOL;
	PB_Cooling_Fan_Request		:	BOOL;
	qq_Spare_1_3				:	BOOL;
	qq_Spare_1_4				:	BOOL;
	qq_Spare_1_5				:	BOOL;
	qq_Spare_1_6				:	BOOL;
	qq_Spare_1_7				:	BOOL;
	
	RAW_Pack_1_Balancing_Amps 	:	BYTE := 20; // 100mA per Bit
	RAW_Pack_2_Balancing_Amps 	:	BYTE := 20; // 100mA per Bit
	RAW_Pack_1_Offset_Volts	  	:	BYTE := 40; // 100mV per Bit
	RAW_Pack_2_Offset_Volts   	:	BYTE := 40; // 100mV per Bit
	qu8_HMI_Spare_6				:	BYTE;
	SW_ePTO_Toggle				:	BOOL;
	ePTO_Speed_Command			:	BYTE;
END_VAR

(* From HMI *)
HMI_Commands_Rx(u32_COBID	:=	16#57B,
				q_NewData => ,
				au8_Data  => ,
				u8_Length => 	);   (*8*)
				
EStop_Bad					:=	HMI_Commands_Rx.au8_Data[0].0;
Hand_Brake_On				:=	HMI_Commands_Rx.au8_Data[0].1;
Heater_Enable				:=	HMI_Commands_Rx.au8_Data[0].2;
StopChargeRq				:=	HMI_Commands_Rx.au8_Data[0].3;
Heater_Low					:=	HMI_Commands_Rx.au8_Data[0].4;
Heater_Med					:=	HMI_Commands_Rx.au8_Data[0].5;
Heater_Hi					:=	HMI_Commands_Rx.au8_Data[0].6;
SW_Isolation_On				:=	HMI_Commands_Rx.au8_Data[0].7;

PB_BMS1_DTC_Reset			:=	HMI_Commands_Rx.au8_Data[1].0;
PB_BMS2_DTC_Reset			:=	HMI_Commands_Rx.au8_Data[1].1;
PB_Cooling_Fan_Request		:=	HMI_Commands_Rx.au8_Data[1].2;
qq_Spare_1_3				:=	HMI_Commands_Rx.au8_Data[1].3;
qq_Spare_1_4				:=	HMI_Commands_Rx.au8_Data[1].4;
qq_Spare_1_5				:=	HMI_Commands_Rx.au8_Data[1].5;
qq_Spare_1_6				:=	HMI_Commands_Rx.au8_Data[1].6;
qq_Spare_1_7				:=	HMI_Commands_Rx.au8_Data[1].7;
	
RAW_Pack_1_Balancing_Amps	:=	HMI_Commands_Rx.au8_Data[2]; 	// WIP
RAW_Pack_2_Balancing_Amps	:=	HMI_Commands_Rx.au8_Data[3];	// WIP
RAW_Pack_1_Offset_Volts		:=	HMI_Commands_Rx.au8_Data[4];	// WIP
RAW_Pack_2_Offset_Volts		:=	HMI_Commands_Rx.au8_Data[5];	// WIP
qu8_HMI_Spare_6				:=	HMI_Commands_Rx.au8_Data[6];
SW_ePTO_Toggle				:=	HMI_Commands_Rx.au8_Data[6].0;	 // Toggle ePTO | TRUE = ON | FALSE = OFF
ePTO_Speed_Command			:=	HMI_Commands_Rx.au8_Data[7]; 	//0.5%/bit

END_PROGRAM

// Application/UserCode/MCU/Dennis_Regen_1
PROGRAM Dennis_Regen_1
VAR
	DennisRegen: CTUD;
	RegenCounterValue: WORD := 4;
END_VAR

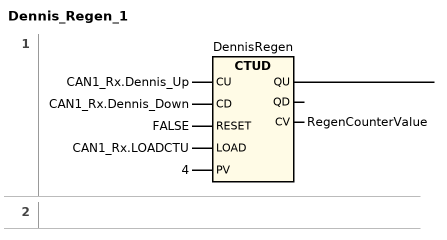
// NETWORK 1
DennisRegen(
    CU := CAN1_Rx.Dennis_Up,
    CD := CAN1_Rx.Dennis_Down,
    RESET := FALSE,
    LOAD := CAN1_Rx.LOADCTU,
    PV := 4,
    CV => RegenCounterValue); // CTUD

// NETWORK 2

END_PROGRAM

// Application/UserCode/MCU/Driveability_1
PROGRAM Driveability_1
VAR
	hq_RegenAvailable	:	BOOL;
	hton_RegenHysteresis	:	TON;
	hr_DriveSpeed	:	REAL;
	hr_FrontSpeed	:	REAL;
	hr_LeftWheels_Speed	:	REAL;
	hr_RightWheels_Speed	:	REAL;
	hr_TractionSpdDiff	:	REAL;
	hr_StabilitySpdDiff	:	REAL;
	
	(*Traction and Stability Dennis and Iveco*)
	TRACTIONLOSS_RELSPEED	:	REAL	:=	300; (*Temporarily set high until time to configure these to the correct value*)
	STABLOSS_RELSPEED		:	REAL	:=	3; (*Temporarily set high until time to configure these to the correct value*)
	(*Bob traction and stability values*)
	TRACTIONLOSS_SPEED	:	UINT	:=	3500;
	STABLOSS_SPEED		:	UINT	:=	1000;
	
	REGEN_CUTOFF_SPEED	:	USINT	:=	5;
	REGEN_WINDDOWNABOVECUTOFF_SPEED	:	USINT	:=	25;
	hton_RegenStartTimer : TON;
	// This ideally should be set to 100ms
	htime_RegenIntro : TIME := T#100MS;
	
	DENNIS_ADJUSTABLE_REGEN	:	REAL	:=	0.4 (*0.4*);
	
	hr_StabilityRelativeDifference : REAL;
	hu8_StabRampSpeed	:	USINT	:=	30;
	hr_STABLOSS_HIGHSPD	:	REAL	:=	2.5;
	hr_StabIncreaseMultiplier	:	REAL	:=	3;
	hr_STABLOSS_HIGHSPD_IVECO	:	REAL	:=	1.5;
	hr_StabIncreaseMultiplier_IVECO	:	REAL	:=	2;
	
	hr_RegenTest	:	REAL	:=	1; (*Use this value in place of the constants for regen multiplier to allow changes to be made by forcing on the fly*)
	
	SecretTractionOff: BOOL;
	hton_Overspeed_Regen: TON;
END_VAR


(*ABS*)
IF (CAN3_Rx.Mode_Button AND CAN3_Rx.Down_Button) = TRUE THEN
	SecretTractionOff :=	TRUE;
END_IF

IF (CAN3_Rx.Mode_Button AND CAN3_Rx.Up_Button) = TRUE THEN
	SecretTractionOff := 	FALSE;
END_IF

IF (gq_ABSActive = TRUE) THEN
	gq_ABS_TorqueDisable	:=	TRUE;
ELSIF (gq_ABSActive = FALSE AND gr_AccelPedal_Perc > 0.03(*3%*)) THEN
	gq_ABS_TorqueDisable	:=	FALSE;
END_IF

IF (gq_Frosty_NoWheelSpeedSensors = TRUE) THEN
	hr_STABLOSS_HIGHSPD_IVECO	:=	10; (*Set so that Stability loss detection does not prevent drive*)
END_IF

IF (gu8_ChassisType = CHASSIS_IVECO AND gq_StabTracDisable_Rx = FALSE) THEN
	(*Traction Control*)
	gr_RearAxle_RelativeSpeed_kph	:= (gr_EBC2_KB_RearRight1RelSpd + gr_EBC2_KB_RearLeft1RelSpd) / 2;
	IF (ABS(gr_RearAxle_RelativeSpeed_kph) > TRACTIONLOSS_RELSPEED(*Change this value to be whatever the speed difference needs to be to trigger can be decimal*)) THEN
		gu8_TractionLoss	:=	1(*TRUE*);
	ELSE
		gu8_TractionLoss	:=	0(*FALSE*);
	END_IF

	(*Stability*)
	IF (gr_VehicleSpeed_kmph > hu8_StabRampSpeed) THEN
		STABLOSS_RELSPEED := hr_STABLOSS_HIGHSPD_IVECO;
	ELSE
		STABLOSS_RELSPEED := hr_STABLOSS_HIGHSPD_IVECO + ((hu8_StabRampSpeed - ABS(gr_VehicleSpeed_kmph)) * hr_StabIncreaseMultiplier_IVECO / hu8_StabRampSpeed);
	END_IF
	
	gr_LeftWheels_RelativeSpeed_kph		:=	(gr_EBC2_KB_FrontLeftRelSpd + gr_EBC2_KB_RearLeft1RelSpd) / 2;
	gr_RightWheels_RelativeSpeed_kph	:=	(gr_EBC2_KB_FrontRightRelSpd + gr_EBC2_KB_RearRight1RelSpd) / 2;
	IF (ABS(gr_LeftWheels_RelativeSpeed_kph) > STABLOSS_RELSPEED OR ABS(gr_RightWheels_RelativeSpeed_kph) > STABLOSS_RELSPEED) THEN (*Can equally use decimal numbers here if needed*)
		gu8_StabilityLoss	:=	1(*TRUE*);
	ELSE
		gu8_StabilityLoss	:=	0(*FALSE*);
	END_IF
ELSIF (gu8_ChassisType = CHASSIS_BOB OR gu8_ChassisType = CHASSIS_ESTARGLIDER) AND (gq_StabTracDisable_Rx = FALSE AND SecretTractionOff = FALSE) THEN // OR should be AND
	(*Traction Control*)
	hr_DriveSpeed	:= (gu16_Bob_RightDrive_CAN + gu16_Bob_LeftDrive_CAN) / 2;
	hr_FrontSpeed	:= (gu16_Bob_RightFront_CAN + gu16_Bob_LeftFront_CAN) / 2;
	hr_TractionSpdDiff	:=	ABS(hr_DriveSpeed - hr_FrontSpeed);
	IF (hr_TractionSpdDiff > TRACTIONLOSS_SPEED(*Change this value to be whatever the speed difference needs to be to trigger can be decimal*)) THEN
		gu8_TractionLoss	:=	1(*TRUE*);
	ELSE
		gu8_TractionLoss	:=	0(*FALSE*);
	END_IF
	(*Stability*)
	hr_LeftWheels_Speed		:=	(gu16_Bob_LeftFront_CAN + gu16_Bob_LeftDrive_CAN) / 2;
	hr_RightWheels_Speed	:=	(gu16_Bob_RightFront_CAN + gu16_Bob_RightDrive_CAN) / 2;
	hr_StabilitySpdDiff		:=	ABS(hr_LeftWheels_Speed - hr_RightWheels_Speed);
	IF (hr_StabilitySpdDiff > STABLOSS_SPEED) THEN (*Can equally use decimal numbers here if needed*)
		gu8_StabilityLoss	:=	1(*TRUE*);
	ELSE
		gu8_StabilityLoss	:=	0(*FALSE*);
	END_IF
ELSIF (gu8_ChassisType = CHASSIS_DENNIS AND (gq_StabTracDisable_Rx = FALSE AND SecretTractionOFF = FALSE)) THEN
	(*Traction Control*)
	(*gr_RearAxle_RelativeSpeed_kph	:= (gr_EBC2_KB_RearRight1RelSpd + gr_EBC2_KB_RearLeft1RelSpd) / 2;
	IF (ABS(gr_RearAxle_RelativeSpeed_kph) > TRACTIONLOSS_RELSPEED(*Change this value to be whatever the speed difference needs to be to trigger can be decimal*)) THEN
		gu8_TractionLoss	:=	1(*TRUE*);
	ELSE
		gu8_TractionLoss	:=	0(*FALSE*);
	END_IF*)
	(*Stability*)
	IF (gr_VehicleSpeed_kmph > hu8_StabRampSpeed) THEN
		STABLOSS_RELSPEED := hr_STABLOSS_HIGHSPD;
	ELSE
		STABLOSS_RELSPEED := hr_STABLOSS_HIGHSPD + ((hu8_StabRampSpeed - ABS(gr_VehicleSpeed_kmph)) * hr_StabIncreaseMultiplier / hu8_StabRampSpeed);
	END_IF
	
	gr_LeftWheels_RelativeSpeed_kph		:=	(gr_EBC2_KB_FrontLeftRelSpd + gr_EBC2_KB_RearLeft1RelSpd) / 2;
	gr_RightWheels_RelativeSpeed_kph	:=	(gr_EBC2_KB_FrontRightRelSpd + gr_EBC2_KB_RearRight1RelSpd) / 2;
	hr_StabilityRelativeDifference	:=	ABS(gr_LeftWheels_RelativeSpeed_kph - gr_RightWheels_RelativeSpeed_kph);
	IF (*(ABS(gr_LeftWheels_RelativeSpeed_kph) > STABLOSS_RELSPEED OR ABS(gr_RightWheels_RelativeSpeed_kph) > STABLOSS_RELSPEED)*)
		(hr_StabilityRelativeDifference > STABLOSS_RELSPEED) THEN (*Can equally use decimal numbers here if needed*)
		gu8_StabilityLoss	:=	1(*TRUE*);
	ELSE
		gu8_StabilityLoss	:=	0(*FALSE*);
	END_IF
	gu8_TractionLoss	:=	gu8_EBC1_ASREngineControlActive;
	(*gu8_StabilityLoss	:=	gu8_EBC1_ASRBrakeControlActive;*)
ELSIF (gq_StabTracDisable_Rx = TRUE) THEN
	gu8_TractionLoss	:=	0(*FALSE*);
	gu8_StabilityLoss	:=	0(*FALSE*);
END_IF


(*Zero torque and Recovery*)
IF (gu8_TractionLoss = 1 OR gu8_StabilityLoss = 1 (* REAMED by IAIN 121021 OR Sevcon2_Control.NO_OIL*)) THEN
	gq_ZeroTorqueRq	:=	TRUE;
	gton_TorqueReIntro_Timer(IN := FALSE, PT := T#0MS);
ELSE
	gton_TorqueReIntro_Timer(IN := TRUE, PT := T#2000MS);
END_IF
IF (gton_TorqueReIntro_Timer.Q = TRUE) THEN
	gq_ZeroTorqueRq	:=	FALSE;
END_IF
gr_TorqueReIntro	:=	TIME_TO_REAL(gton_TorqueReIntro_Timer.ET);
gr_TorqueReIntroMax	:=	TIME_TO_REAL(T#2000MS);

(*Regen*)
(*Selectable regen setting needed*)
IF (gu8_BMS_SOC < 90) THEN
	gr_RegenSOCMultiplier	:=	1;
ELSIF (gu8_BMS_SOC >= 90 AND gu8_BMS_SOC < 95) THEN
	gr_RegenSOCMultiplier	:=	0.5;
ELSE
	gr_RegenSOCMultiplier	:=	0;
END_IF


IF (gr_VehicleSpeed_kmph > REGEN_CUTOFF_SPEED) THEN
	hton_RegenHysteresis(IN := TRUE, PT := T#1000MS); // bring down to T#1s? Was t#5s
ELSE
	hton_RegenHysteresis(IN := FALSE, PT := T#0S);
END_IF
hq_RegenAvailable	:=	hton_RegenHysteresis.Q;

hton_Overspeed_Regen (IN:= gr_VehicleSpeed_kmph > 55, PT:= T#5S);
IF ((gr_AccelPedal_Perc < 0.01 OR (gr_VehicleSpeed_kmph > 55 AND hton_Overspeed_Regen.Q)) AND hq_RegenAvailable = TRUE) THEN //OR gr_VehicleSpeed_kmph > 56 added
	gq_RegenActive	:=	TRUE;
	gr_RegenSpeedDegrading	:=	LIMIT(0, (gr_VehicleSpeed_kmph - REGEN_CUTOFF_SPEED), REGEN_WINDDOWNABOVECUTOFF_SPEED) / REGEN_WINDDOWNABOVECUTOFF_SPEED;
	IF gr_VehicleSpeed_kmph > 55 THEN
	DENNIS_ADJUSTABLE_REGEN := 1.2;
	END_IF
//////////////	

//DENNIS with BRAKE
	IF (gu8_ChassisType = CHASSIS_DENNIS AND gq_BrakeSwitch = TRUE) THEN
		DENNIS_ADJUSTABLE_REGEN := 1.2;
		gr_RegenMultiplierRq	:=	DENNIS_ADJUSTABLE_REGEN;
		hton_RegenStartTimer(IN := TRUE, PT := htime_RegenIntro);
		gr_RegenIntroCF := LIMIT(0, (TIME_TO_REAL(hton_RegenStartTimer.ET) / TIME_TO_REAL(hton_RegenStartTimer.PT)), 1);
	END_IF
//DENNIS without BRAKE	
	IF (gu8_ChassisType = CHASSIS_DENNIS AND gq_BrakeSwitch = FALSE) THEN
		gr_RegenMultiplierRq	:=	DENNIS_ADJUSTABLE_REGEN(*40%*);
		hton_RegenStartTimer(IN := TRUE, PT := htime_RegenIntro);
		gr_RegenIntroCF := LIMIT(0, (TIME_TO_REAL(hton_RegenStartTimer.ET) / TIME_TO_REAL(hton_RegenStartTimer.PT)), 1);
		
		IF Dennis_Regen.RegenCounterValue = 0 THEN 
			DENNIS_ADJUSTABLE_REGEN := 0;
		END_IF
		IF Dennis_Regen.RegenCounterValue = 1 THEN
			DENNIS_ADJUSTABLE_REGEN := 0.6;
		END_IF
		IF Dennis_Regen.RegenCounterValue = 2 THEN
			DENNIS_ADJUSTABLE_REGEN := 0.8;
		END_IF
		IF Dennis_Regen.RegenCounterValue = 3 THEN
			DENNIS_ADJUSTABLE_REGEN := 1;
		END_IF
		IF Dennis_Regen.RegenCounterValue = 4 THEN
			DENNIS_ADJUSTABLE_REGEN := 1.2;
		END_IF	
//////////////		

ELSIF (gq_BrakeSwitch = TRUE AND gu8_ChassisType <> CHASSIS_DENNIS) THEN
		IF (gu8_RegenSelector = 0) THEN
			gr_RegenMultiplierRq	:=	0.7(*40%*);
			hton_RegenStartTimer(IN := TRUE, PT := htime_RegenIntro);
			gr_RegenIntroCF := LIMIT(0, (TIME_TO_REAL(hton_RegenStartTimer.ET) / TIME_TO_REAL(hton_RegenStartTimer.PT)), 1);
		ELSIF (gu8_RegenSelector = 1) THEN
			gr_RegenMultiplierRq	:=	0.7(*40%*);
			hton_RegenStartTimer(IN := TRUE, PT := htime_RegenIntro);
			gr_RegenIntroCF := LIMIT(0, (TIME_TO_REAL(hton_RegenStartTimer.ET) / TIME_TO_REAL(hton_RegenStartTimer.PT)), 1);
		ELSIF (gu8_RegenSelector = 2) THEN
			gr_RegenMultiplierRq	:=	0.7(*60%*);
			hton_RegenStartTimer(IN := TRUE, PT := htime_RegenIntro);
			gr_RegenIntroCF := LIMIT(0, (TIME_TO_REAL(hton_RegenStartTimer.ET) / TIME_TO_REAL(hton_RegenStartTimer.PT)), 1);
		END_IF
	ELSIF (gq_BrakeSwitch = FALSE AND gu8_ChassisType <> CHASSIS_DENNIS) THEN
		IF (gu8_RegenSelector = 0) THEN
			gr_RegenMultiplierRq	:=	0(*0%*);
			hton_RegenStartTimer(IN := FALSE, PT := T#0MS);
			gr_RegenIntroCF := 0;
		ELSIF (gu8_RegenSelector = 1) THEN
			gr_RegenMultiplierRq	:=	0.6(*0.4(*40%*)*);
			hton_RegenStartTimer(IN := TRUE, PT := htime_RegenIntro);
			gr_RegenIntroCF := LIMIT(0, (TIME_TO_REAL(hton_RegenStartTimer.ET) / TIME_TO_REAL(hton_RegenStartTimer.PT)), 1);
		ELSIF (gu8_RegenSelector = 2) THEN
			gr_RegenMultiplierRq	:=	1(*0.6(*60%*)*);
			hton_RegenStartTimer(IN := TRUE, PT := htime_RegenIntro);
			gr_RegenIntroCF := LIMIT(0, (TIME_TO_REAL(hton_RegenStartTimer.ET) / TIME_TO_REAL(hton_RegenStartTimer.PT)), 1);
		END_IF
	END_IF
ELSE
	gq_RegenActive	:=	FALSE;
	gr_RegenMultiplierRq	:=	0;
	hton_RegenStartTimer(IN := FALSE, PT := T#0MS);
	gr_RegenIntroCF := 0;
END_IF
(*Also need battery SOC as multiplier <90 x1, 90<X<95 x0.5, >95 x0*)





(*Creep / Hill hold*)

END_PROGRAM

// Application/UserCode/MCU/f_DistanceCalc_1
FUNCTION f_DistanceCalc_1 : REAL
VAR_INPUT
	gr_MotorRotation_IN		:	REAL;
	gu16_GearRatio_IN		:	UINT;
	gu16_DyfRatio_IN		:	UINT;
	gu16_TireWidth_IN		:	UINT;
	gu8_TireProfile_IN		:	USINT;
	gu16_WheelDiameter_IN	:	UINT;
END_VAR
VAR
	hr_SidewallWidth_m	:	REAL;
	hr_TotalWheelDiameter_m	:	REAL;
	hr_WheelCircumfrence_km	:	REAL;
	hr_RevsPerKm			:	REAL;
	
	hr_GearRatio				:	REAL;
	hr_DyfRatio					:	REAL;
	hr_WheelDiameter_inch		:	REAL;
	hr_WheelDiameter_m			:	REAL;
END_VAR
VAR CONSTANT
	PI	:	REAL	:=	3.14159;
	INCH_TO_METER_CF	:	REAL	:=	0.0254;
	MILLI_TO_METER		:	UINT	:=	1000;
END_VAR


hr_GearRatio				:=	gu16_GearRatio_IN / 1000;
hr_DyfRatio					:=	gu16_DyfRatio_IN / 1000;
hr_WheelDiameter_inch		:=	gu16_WheelDiameter_IN / 10;

hr_WheelDiameter_m			:=	hr_WheelDiameter_inch * INCH_TO_METER_CF;
hr_SidewallWidth_m			:=	gu16_TireWidth_mm * (gu8_TireProfile_Perc / 100) / MILLI_TO_METER;
hr_TotalWheelDiameter_m		:=	hr_WheelDiameter_m + hr_SidewallWidth_m;

hr_WheelCircumfrence_km		:=	(hr_TotalWheelDiameter_m * PI) / 1000;
hr_RevsPerKm				:=	1 / hr_WheelCircumfrence_km;

f_DistanceCalc	:=	gr_MotorRotation_IN / hr_GearRatio / hr_DyfRatio / hr_RevsPerKm;

END_FUNCTION

// Application/UserCode/MCU/f_SpeedCalc_1
FUNCTION f_SpeedCalc_1 : REAL
VAR_INPUT
	gr_MotorSpeed_IN		:	REAL;
	gu16_GearRatio_IN		:	UINT;
	gu16_DyfRatio_IN		:	UINT;
	gu16_TireWidth_IN		:	UINT;
	gu8_TireProfile_IN		:	USINT;
	gu16_WheelDiameter_IN	:	UINT;
END_VAR
VAR
	hr_SidewallWidth_m	:	REAL;
	hr_TotalWheelDiameter_m	:	REAL;
	hr_WheelCircumfrence_km	:	REAL;
	hr_RevsPerKm			:	REAL;
	
	hr_GearRatio				:	REAL;
	hr_DyfRatio					:	REAL;
	hr_WheelDiameter_inch		:	REAL;
	hr_WheelDiameter_m			:	REAL;
END_VAR
VAR CONSTANT
	PI	:	REAL	:=	3.14159;
	INCH_TO_METER_CF	:	REAL	:=	0.0254;
	MILLI_TO_METER		:	UINT	:=	1000;
END_VAR


hr_GearRatio				:=	gu16_GearRatio_IN / 1000;
hr_DyfRatio					:=	gu16_DyfRatio_IN / 1000;
hr_WheelDiameter_inch		:=	gu16_WheelDiameter_IN / 10;

hr_WheelDiameter_m			:=	hr_WheelDiameter_inch * INCH_TO_METER_CF;
hr_SidewallWidth_m			:=	gu16_TireWidth_mm * (gu8_TireProfile_Perc / 100) / MILLI_TO_METER;
hr_TotalWheelDiameter_m		:=	hr_WheelDiameter_m + hr_SidewallWidth_m;

hr_WheelCircumfrence_km		:=	(hr_TotalWheelDiameter_m * PI) / 1000;
hr_RevsPerKm				:=	1 / hr_WheelCircumfrence_km;

f_SpeedCalc	:=	gr_MotorSpeed_IN / hr_GearRatio / hr_DyfRatio / hr_RevsPerKm * 60;

END_FUNCTION

// Application/UserCode/MCU/GearSelection_1
PROGRAM GearSelection_1
VAR
END_VAR

(*Do I need to ensure low speed for gear change*)
(*ADDED minimal vehicle speed to gear selection*)

IF (gu8_SystemState = DRIVE_SYS AND DO_q_BatteryDischargeMain_DO = TRUE) THEN
	IF (gq_Gear_Drive_Rq = TRUE AND gq_BrakeSwitch = TRUE) AND gr_VehicleSpeed_kmph > -1 THEN
		gq_Gear_Neutral			:=	FALSE;
		gq_Gear_Drive			:=	TRUE;
		gq_Gear_DriveCrawl		:=	FALSE;
		gq_Gear_Reverse			:=	FALSE;
		gq_Gear_ReverseCrawl	:=	FALSE; (*Select Drive*)
	ELSIF (gq_Gear_Neutral_Rq = TRUE AND gq_BrakeSwitch = TRUE) AND (gr_VehicleSpeed_kmph <1 AND gr_VehicleSpeed_kmph >-1) THEN
		gq_Gear_Neutral			:=	TRUE;
		gq_Gear_Drive			:=	FALSE;
		gq_Gear_DriveCrawl		:=	FALSE;
		gq_Gear_Reverse			:=	FALSE;
		gq_Gear_ReverseCrawl	:=	FALSE; (*Select Neutral*)
	ELSIF (gq_Gear_Reverse_Rq = TRUE AND gq_BrakeSwitch = TRUE) AND gr_VehicleSpeed_kmph < 1 THEN
		gq_Gear_Neutral			:=	FALSE;
		gq_Gear_Drive			:=	FALSE;
		gq_Gear_DriveCrawl		:=	FALSE;
		gq_Gear_Reverse			:=	TRUE;
		gq_Gear_ReverseCrawl	:=	FALSE; (*Select Reverse*)
	ELSIF (DI_q_DirectionSwitch_DriveCrawl_DI = TRUE AND gq_BrakeSwitch = TRUE) THEN
		gq_Gear_Neutral			:=	FALSE;
		gq_Gear_Drive			:=	FALSE;
		gq_Gear_DriveCrawl		:=	TRUE;
		gq_Gear_Reverse			:=	FALSE;
		gq_Gear_ReverseCrawl	:=	FALSE; (*Select Drive Crawl*)
	(*ELSIF (DI_q_DirectionSwitch_ReverseCrawl_DI = TRUE AND gq_BrakeSwitch = TRUE) THEN
		gq_Gear_Neutral			:=	FALSE;
		gq_Gear_Drive			:=	FALSE;
		gq_Gear_DriveCrawl		:=	FALSE;
		gq_Gear_Reverse			:=	FALSE;
		gq_Gear_ReverseCrawl	:=	TRUE; (*Select Reverse Crawl*)*)
	END_IF
ELSIF (gu8_SystemState <> DRIVE_SYS) THEN
	gq_Gear_Neutral			:=	TRUE;
	gq_Gear_Drive			:=	FALSE;
	gq_Gear_DriveCrawl		:=	FALSE;
	gq_Gear_Reverse			:=	FALSE;
	gq_Gear_ReverseCrawl	:=	FALSE; (*Gear selection = Neutral*)
ELSE
	gq_Gear_Neutral			:=	TRUE;
	gq_Gear_Drive			:=	FALSE;
	gq_Gear_DriveCrawl		:=	FALSE;
	gq_Gear_Reverse			:=	FALSE;
	gq_Gear_ReverseCrawl	:=	FALSE; (*Neutral*)
END_IF

gq_ReverseLights	:=	gq_Gear_Reverse;

END_PROGRAM

// Application/UserCode/MCU/MCU_Control_1
PROGRAM MCU_Control_1
VAR
	hs8_Direction	:	SINT	:=	0;
	hton_Mileometer	:	TON;
	hq_SetInitialDistance	:	BOOL	:=	FALSE;
	hton_TorqueRqRamp	:	TON;
	hr_TorqueRampTime	:	REAL;
	hr_TorqueRampTotal	:	REAL;
	hr_MCU_TorquePreRamp	:	REAL;
	hf_TorqueRamp			:	Ramp_Linear;
	
	TORQUE_RQ_CF	:	REAL	:=	0.3; (*In case any conversion factors need to be applied to the value being sent*)
	hr_MULTIPLIER_CALC	: REAL	:= 0;
	WINDUPSPEED			: USINT := 10;
	
	hr_SpeedLimit_KP	:	REAL	:=	10;
	hr_SpeedLimit_KI	:	REAL	:=	10;
	hfb_SpeedLimit_PID	:	PID;
	hr_MaximumTorqueLimit : REAL;
	hr_TARGETMAXSPEED : REAL := 77;
	hr_IntegralCounter : ARRAY [0..49] OF REAL;
	Counter : USINT := 0;
	hr_IntegralSum : REAL := 0;
	Cycle : USINT;
END_VAR
VAR CONSTANT
	INITIALISATION	:	USINT	:=	0;
	STANDBY			:	USINT	:=	1;
	STARTUP			:	USINT	:=	2;
	TEARDOWN		:	USINT	:=	3;
	OPERATIONAL		:	USINT	:=	4;
	FAILURE			:	USINT	:=	5;
	CLOSEDOWN		:	USINT	:=	6;
	READYTOSHUTDOWN	:	USINT	:=	7;
	WAITFORCOOLING	:	USINT	:=	8;
	
	SHUTDOWN_RQ		:	USINT	:=	2;
	OPERATIONAL_RQ	:	USINT	:=	1;
	STANDBY_RQ		:	USINT	:=	0;
	
	TORQUE_MODE		:	USINT	:=	1;
	SPEED_MODE		:	USINT	:=	2;
	
	
	
	EV_MODE			:	USINT	:=	3;
	NEU_NOTORQUE	:	USINT	:=	0;

END_VAR

IF (DI_q_VehicleKL15_DI = TRUE) THEN
	hton_Mileometer(IN := TRUE, PT := T#60S);
	IF (gu16_MCU_MaxMotorSpeed_Rx = 0) THEN
		gu8_MCU_VMUPollMCU_Multiplex	:=	MAXMOTORSPEED;
	ELSIF (gu16_MCU_MaxMotorTorque_Rx = 0) THEN
		gu8_MCU_VMUPollMCU_Multiplex	:=	MAXMOTORTORQUE;
	ELSIF (hton_Mileometer.Q = TRUE) THEN
		hton_Mileometer(IN := FALSE, PT := T#0S);
		gu8_MCU_VMUPollMCU_Multiplex	:=	TOTALMOTORROTATION;
	ELSE
		gu8_MCU_VMUPollMCU_Multiplex	:=	8; (*Not applicable value so will not incorrectly request any data*)
	END_IF
END_IF

(*Must be in discharge mode and precharge complete before command out of standby (Need to set ignition at the start always)*)
IF (gu8_SystemState = DRIVE_SYS AND DOS_q_BatteryDischargeMain_DO = TRUE(* AND gr_MCU_TractionTorqueAvailable > 0*)) THEN
	IF ((gu8_MCU_State = STANDBY) AND gq_Gear_Neutral = TRUE) THEN
		gu8_MCU_OperationRequest	:=	OPERATIONAL_RQ;
		gu8_MCU_OperationalMode_Tx	:=	NEU_NOTORQUE;
	ELSIF (gu8_MCU_State = OPERATIONAL) THEN
		gu8_MCU_OperationRequest	:=	OPERATIONAL_RQ;
		gu8_MCU_OperationalMode_Tx	:=	EV_MODE;
	END_IF
ELSIF (gu8_SystemState <> DRIVE_SYS) THEN
	IF (gu8_MCU_State = OPERATIONAL AND gq_Gear_Neutral = TRUE) THEN
		gu8_MCU_OperationRequest	:=	SHUTDOWN_RQ;
		gu8_MCU_OperationalMode_Tx	:=	NEU_NOTORQUE;
	ELSIF (gu8_MCU_State = OPERATIONAL AND gq_Gear_Neutral = FALSE) THEN
		gu8_MCU_OperationRequest	:=	OPERATIONAL_RQ;
		gu8_MCU_OperationalMode_Tx	:=	NEU_NOTORQUE;
		(*Rq Neutral*)
	ELSE
		gu8_MCU_OperationRequest	:=	STANDBY_RQ;
		gu8_MCU_OperationalMode_Tx	:=	NEU_NOTORQUE;
	END_IF
ELSE
	gu8_MCU_OperationRequest	:=	STANDBY_RQ;
	gu8_MCU_OperationalMode_Tx	:=	NEU_NOTORQUE;
END_IF

(*These values should be set by the BMS*)
gu16_MCU_MaxChargeCurrent		:=	REAL_TO_UINT(gr_BMS_CCL);
gu16_MCU_MaxDischargeCurrent	:=	REAL_TO_UINT(gr_BMS_DCL);
gu16_MCU_MaxBatteryVoltage		:=	gu16_BMS_Maximum_Pack_Voltage;
gu16_MCU_MinBatteryVoltage		:=	gu16_BMS_MinimumPackVoltage;
gu8_MCU_CommandMode				:=	TORQUE_MODE;
gu8_MCU_ReferenceCommandMode	:=	TORQUE_MODE;
gr_MCU_MaxMotorSpeed_PreCF		:=	gr_MCU_MaxMotorSpeed; (*This may need to be set for safety*)

IF (gq_Gear_Drive = TRUE OR gq_Gear_DriveCrawl = TRUE) THEN
	hs8_Direction	:=	1;
	gq_MCU_SpeedCommandStatus		:=	FALSE;
	gq_MCU_TorqueCommandStatus		:=	FALSE;
ELSIF (gq_Gear_Reverse = TRUE OR gq_Gear_ReverseCrawl = TRUE) THEN
	hs8_Direction	:=	-1;
	gq_MCU_SpeedCommandStatus		:=	FALSE;
	gq_MCU_TorqueCommandStatus		:=	FALSE;
ELSE
	hs8_Direction	:=	0;
	gq_MCU_SpeedCommandStatus		:=	TRUE;
	gq_MCU_TorqueCommandStatus		:=	TRUE;
END_IF

hr_MULTIPLIER_CALC := gr_VehicleSpeed_kmph / WINDUPSPEED;
TORQUE_RQ_CF := LIMIT(1(*0.3*), hr_MULTIPLIER_CALC, 1);

Driveability();
IF (gu8_MCU_State = OPERATIONAL AND hs8_Direction <> 0 (*Not in neutral*) AND gq_ABSActive = FALSE AND gq_BodySteps = FALSE) THEN
	IF (gq_ABS_TorqueDisable = TRUE) THEN
		hton_TorqueRqRamp(IN := FALSE, PT := T#0S);
		gr_MCU_TorqueCommand_PreCF			:=	0;
	ELSIF (gq_ZeroTorqueRq = TRUE) THEN
		hton_TorqueRqRamp(IN := FALSE, PT := T#0S);
		IF (gq_RegenActive = TRUE) THEN
			gr_MCU_TorqueCommand_PreCF	:=	(*gr_MCU_MaxMotorTorque*)gr_MCU_RegenTorqueAvailable * gr_RegenSOCMultiplier * gr_RegenMultiplierRq * gr_RegenSpeedDegrading * gr_RegenIntroCF * (hs8_Direction * (-1)) * LIMIT(0, (gr_TorqueReIntro / gr_TorqueReIntroMax), 1);(**)
		ELSIF (gq_RegenActive = FALSE) THEN
			gr_MCU_TorqueCommand_PreCF			:=	gr_AccelPedal_Perc * TORQUE_RQ_CF * hs8_Direction * (*gr_MCU_MaxMotorTorque*)gr_MCU_TractionTorqueAvailable * LIMIT(0, (gr_TorqueReIntro / gr_TorqueReIntroMax), 1);
		END_IF
	ELSIF (gq_ABS_TorqueDisable = FALSE AND gq_ZeroTorqueRq = FALSE) THEN
		IF (gq_RegenActive = TRUE) THEN
			hton_TorqueRqRamp(IN := FALSE, PT := T#0S);
			gr_MCU_TorqueCommand_PreCF	:=	(*gr_MCU_MaxMotorTorque*)gr_MCU_RegenTorqueAvailable * gr_RegenSOCMultiplier * gr_RegenMultiplierRq * gr_RegenSpeedDegrading * gr_RegenIntroCF * (hs8_Direction * (-1));(**)
		ELSIF (gq_RegenActive = FALSE) THEN	
			hr_MCU_TorquePreRamp	:=	gr_AccelPedal_Perc * TORQUE_RQ_CF * hs8_Direction * (*gr_MCU_MaxMotorTorque*)gr_MCU_TractionTorqueAvailable;
			gr_MCU_TorqueCommand_PreCF	:=	hr_MCU_TorquePreRamp;
		END_IF
	END_IF
	//*DO_q_DrivetrainCoolingFan_DO		:=	TRUE;
ELSE
	gr_MCU_TorqueCommand_PreCF			:=	0 * TORQUE_RQ_CF * (*gr_MCU_MaxMotorTorque*)gr_MCU_TractionTorqueAvailable;
	//*DO_q_DrivetrainCoolingFan_DO		:=	FALSE;
	hton_TorqueRqRamp(IN := FALSE, PT := T#0S);
END_IF

IF (gu8_BMS_SOC > 10) THEN
	IF (gu8_ChassisType <> CHASSIS_IVECO) THEN
		hr_TARGETMAXSPEED := SpeedOTG;
	ELSIF (gu8_ChassisType = CHASSIS_IVECO) THEN
		hr_TARGETMAXSPEED := 55;
	END_IF
ELSE
	IF (gu8_ChassisType <> CHASSIS_IVECO) THEN
		hr_TARGETMAXSPEED := SpeedOTG1;
	ELSIF (gu8_ChassisType = CHASSIS_IVECO) THEN
		hr_TARGETMAXSPEED := 24;
	END_IF
END_IF

IF (gr_VehicleSpeed_kmph > hr_TARGETMAXSPEED) THEN
	hr_MaximumTorqueLimit := 0;
ELSE
	hr_IntegralCounter[Counter] := LIMIT(0, (hr_TARGETMAXSPEED - gr_VehicleSpeed_kmph), hr_TARGETMAXSPEED);
	IF (Counter > 49) THEN
		Counter := 0;
	ELSE
		Counter := Counter + 1;
	END_IF
	hr_IntegralSum := 0;
	FOR Cycle := 0 TO 49 DO
		hr_IntegralSum := hr_IntegralSum + hr_IntegralCounter[Cycle];
	END_FOR
	hr_MaximumTorqueLimit := MAX(((hr_TARGETMAXSPEED - gr_VehicleSpeed_kmph) * hr_SpeedLimit_KP + hr_IntegralSum * hr_SpeedLimit_KI), 0);
END_IF


gr_MCU_SpeedCommand_PreCF			:=	0;

gr_MCU_TorqueCommand_PreCF_Limited	:=	LIMIT(-3500, gr_MCU_TorqueCommand_PreCF, hr_MaximumTorqueLimit);
gr_MCU_ReferenceTorqueCommand_PreCF	:=	LIMIT(-3500, gr_MCU_TorqueCommand_PreCF, hr_MaximumTorqueLimit);
gr_MCU_ReferenceSpeedCommand_PreCF	:=	gr_MCU_SpeedCommand_PreCF;

(*Don't think I need to set these but will keep them here as a reminder and just in case they do need setting*)
gq_MCU_MaxDiscahrgeCurrentStatus	:=	FALSE;
gq_MCU_MaxBatteryVoltageStatus		:=	FALSE;
gq_MCU_MinBatteryVoltageStatus		:=	FALSE;
gq_MCU_MaxChargeCurrentStatus		:=	FALSE;

gr_VehicleSpeed_kmph	:=	f_SpeedCalc(gr_MotorSpeed_IN := gr_MCU_MotorSpeed, gu16_GearRatio_IN := gu16_GearRatio_PreCF,
										gu16_DyfRatio_IN := gu16_DyfRatio_PreCF, gu16_TireWidth_IN := gu16_TireWidth_mm,
										gu8_TireProfile_IN := gu8_TireProfile_Perc, gu16_WheelDiameter_IN := gu16_WheelDiameter_PreCF);

gr_VehicleAllTimeDistance	:=	f_DistanceCalc(gr_MotorRotation_IN := gr_MCU_TotalMotorRotation, gu16_GearRatio_IN := gu16_GearRatio_PreCF,
										gu16_DyfRatio_IN := gu16_DyfRatio_PreCF, gu16_TireWidth_IN := gu16_TireWidth_mm,
										gu8_TireProfile_IN := gu8_TireProfile_Perc, gu16_WheelDiameter_IN := gu16_WheelDiameter_PreCF);

IF (hq_SetInitialDistance = FALSE AND gr_MCU_TotalMotorRotation <> 0) THEN
	gr_VehicleInitialTripDistance	:=	gr_VehicleAllTimeDistance;
	hq_SetInitialDistance			:=	TRUE;
END_IF

gr_VehicleTripDistance	:=	gr_VehicleAllTimeDistance - gr_VehicleInitialTripDistance;

END_PROGRAM

// Application/UserCode/MCU/MCU_Rx_1
PROGRAM MCU_Rx_1
VAR
	MCU_CommandResponse1_Rx		:	Receive_CAN1_STD;
	MCU_CommandResponse2_Rx		:	Receive_CAN1_STD;
	MCU_EventInfo1_Rx			:	Receive_CAN1_STD;
	MCU_Info1_Rx				:	Receive_CAN1_STD;
	MCU_Info2_Rx				:	Receive_CAN1_STD;
	MCU_OnEventInfo1_Rx			:	Receive_CAN1_STD;
	MCU_Thermal1_Rx				:	Receive_CAN1_STD;
	MCU_PollingMCUResponse_Rx	:	Receive_CAN1_STD;
	MCU_PollingVMU_Rx			:	Receive_CAN1_STD;
	
	MCU_CommandResponse1_Rx_Timer	:	TON;
	MCU_CommandResponse2_Rx_Timer	:	TON;
	MCU_EventInfo1_Rx_Timer			:	TON;
	MCU_Info1_Rx_Timer				:	TON;
	MCU_Info2_Rx_Timer				:	TON;
	MCU_Thermal1_Rx_Timer			:	TON;
END_VAR


MCU_CommandResponse1_Rx(u32_COBID	:=	16#043,
						 q_NewData => ,
						 au8_Data => ,
						 u8_Length => 			);
						 
MCU_CommandResponse2_Rx(u32_COBID	:=	16#044,
						 q_NewData => ,
						 au8_Data => ,
						 u8_Length => 			);
						 
MCU_EventInfo1_Rx(u32_COBID	:=	16#442,
						 q_NewData => ,
						 au8_Data => ,
						 u8_Length => 			);
						 
MCU_Info1_Rx(u32_COBID	:=	16#440,
						 q_NewData => ,
						 au8_Data => ,
						 u8_Length => 			);
						 
MCU_Info2_Rx(u32_COBID	:=	16#441,
						 q_NewData => ,
						 au8_Data => ,
						 u8_Length => 			);
						 
MCU_OnEventInfo1_Rx(u32_COBID	:=	16#443,
						 q_NewData => ,
						 au8_Data => ,
						 u8_Length => 			);
						 
MCU_Thermal1_Rx(u32_COBID	:=	16#449,
						 q_NewData => ,
						 au8_Data => ,
						 u8_Length => 			);
						 
MCU_PollingMCUResponse_Rx(u32_COBID	:=	16#448,
						 q_NewData => ,
						 au8_Data => ,
						 u8_Length => 			);
						 
MCU_PollingVMU_Rx(u32_COBID	:=	16#445,
						 q_NewData => ,
						 au8_Data => ,
						 u8_Length => 			);
						 


(*MCUCommandResponse1*)
gu8_MCU_State								:=	MCU_CommandResponse1_Rx.au8_Data[0] AND 2#00001111;
gu8_MCU_OperationalMode						:=	MCU_CommandResponse1_Rx.au8_Data[0] AND 2#01110000;
gq_MCU_RegenDeratingStatus					:=	MCU_CommandResponse1_Rx.au8_Data[0].7;
gu8_MCU_RegenDerating						:=	MCU_CommandResponse1_Rx.au8_Data[1] AND 2#00001111;
gu8_MCU_TractionDerating					:=	MCU_CommandResponse1_Rx.au8_Data[1] AND 2#11110000;
gu16_MCU_MaxMotorSpeedForward_Rx			:=	USINT_TO_UINT(MCU_CommandResponse1_Rx.au8_Data[2]) +
												SHL(BOOL_TO_UINT(MCU_CommandResponse1_Rx.au8_Data[3].0), 8);
gu16_MCU_MaxMotorSpeedReverse_Rx			:=	USINT_TO_UINT(MCU_CommandResponse1_Rx.au8_Data[4]) +
												SHL(BOOL_TO_UINT(MCU_CommandResponse1_Rx.au8_Data[5].0), 8);
gq_MCU_MaxMotorSpeedForwardStatus			:=	MCU_CommandResponse1_Rx.au8_Data[5].1;
gq_MCU_MaxMotorSpeedReverseStatus			:=	MCU_CommandResponse1_Rx.au8_Data[5].2;
gq_MCU_TractionDeratingStatus				:=	MCU_CommandResponse1_Rx.au8_Data[5].3;
gu8_MCU_RollingCounter_Comm1				:=	MCU_CommandResponse1_Rx.au8_Data[5] AND 2#11110000;
(*MCUCommandResponse2*)
gu16_MCU_MotorSpeed_Rx						:=	USINT_TO_UINT(MCU_CommandResponse2_Rx.au8_Data[0]) +
												SHL(USINT_TO_UINT(MCU_CommandResponse2_Rx.au8_Data[1]), 8);
gu16_MCU_MotorAngle_Rx						:=	USINT_TO_UINT(MCU_CommandResponse2_Rx.au8_Data[2]) +
												SHL(USINT_TO_UINT(MCU_CommandResponse2_Rx.au8_Data[3]), 8);
gq_MVU_MotorAngleStatus						:=	MCU_CommandResponse2_Rx.au8_Data[4].0;
gq_MCU_MotorSpeedStatus						:=	MCU_CommandResponse2_Rx.au8_Data[4].1;
gq_MCU_SpeedReductionRequest				:=	MCU_CommandResponse2_Rx.au8_Data[4].2;
gq_MCU_EmergencyStop						:=	MCU_CommandResponse2_Rx.au8_Data[4].3;
gu8_MCU_RollingCounter_Comm2				:=	MCU_CommandResponse2_Rx.au8_Data[4] AND 2#11110000;
(*MCUEventInfo1*)
gq_MCU_Fault_PhaseToChassis					:=	MCU_EventInfo1_Rx.au8_Data[0].0;
gq_MCU_Fault_InterlockBatteryCable			:=	MCU_EventInfo1_Rx.au8_Data[0].1;
gq_MCU_Fault_InterlockMotorCable			:=	MCU_EventInfo1_Rx.au8_Data[0].2;
gq_MCU_Fault_DriveCoverWasOpened			:=	MCU_EventInfo1_Rx.au8_Data[0].3;
gq_MCU_Fault_PhaseToChassisStatus			:=	MCU_EventInfo1_Rx.au8_Data[0].4;
gq_MCU_Fault_InterlockBatteryCableStatus	:=	MCU_EventInfo1_Rx.au8_Data[0].5;
gq_MCU_Fault_InterlockMotorCableStatus		:=	MCU_EventInfo1_Rx.au8_Data[0].6;
gq_MCU_Fault_DriveCoverWasOpenedStatus		:=	MCU_EventInfo1_Rx.au8_Data[0].7;
(*MCUInfo1*)
gu8_MCU_AuxiliaryVoltage_Rx					:=	MCU_Info1_Rx.au8_Data[0];
gu16_MCU_HighPowerVoltage					:=	USINT_TO_UINT(MCU_Info1_Rx.au8_Data[1]) +
												SHL(USINT_TO_UINT(MCU_Info1_Rx.au8_Data[2] AND 2#00000111), 8);
gq_MCU_HighPowerCurrentStatus				:=	MCU_Info1_Rx.au8_Data[2].3;
gq_MCU_AuxiliaryVoltageStatus				:=	MCU_Info1_Rx.au8_Data[2].4;
gq_MCU_HighPowerVoltageStatus				:=	MCU_Info1_Rx.au8_Data[2].5;
gu16_MCU_HighPowerCurrent_Rx				:=	USINT_TO_UINT(MCU_Info1_Rx.au8_Data[3]) +
												SHL(USINT_TO_UINT(MCU_Info1_Rx.au8_Data[4]), 8);
gu8_MCU_RollingCounter_Info1				:=	MCU_Info1_Rx.au8_Data[5];
(*MCUInfo2*)
gu16_MCU_MotorTorqueEstimated_Rx			:=	USINT_TO_UINT(MCU_Info2_Rx.au8_Data[0]) +
												SHL(USINT_TO_UINT(MCU_Info2_Rx.au8_Data[1]), 8);
gu16_MCU_TractionTorqueAvailable_Rx			:=	USINT_TO_UINT(MCU_Info2_Rx.au8_Data[2]) +
												SHL(USINT_TO_UINT(MCU_Info2_Rx.au8_Data[3] AND 2#01111111), 8);
gu16_MCU_RegenTorqueAvailable_Rx			:=	USINT_TO_UINT(MCU_Info2_Rx.au8_Data[4]) +
												SHL(USINT_TO_UINT(MCU_Info2_Rx.au8_Data[5] AND 2#01111111), 8);
gq_MCU_MotorTorqueEstimatedStatus			:=	MCU_Info2_Rx.au8_Data[6].1;
gq_MCU_TractionTorqueAvailableStatus		:=	MCU_Info2_Rx.au8_Data[6].2;
gq_MCU_RegenTorqueAvailableStatus			:=	MCU_Info2_Rx.au8_Data[6].3;
gu8_MCU_RollingCounter_Info2				:=	MCU_Info2_Rx.au8_Data[6] AND 2#11110000;
(*MCUOnEventInfo1*)
gu16_MCU_EventID							:=	USINT_TO_UINT(MCU_OnEventInfo1_Rx.au8_Data[0]) +
												SHL(USINT_TO_UINT(MCU_OnEventInfo1_Rx.au8_Data[1]), 8);
gu8_MCU_RollingCounter_OnEventInfo1			:=	MCU_OnEventInfo1_Rx.au8_Data[4] AND 2#11110000;
(*MCUThermal1*)
gu8_MCU_DriveCoolingFlowRequest_Rx			:=	MCU_Thermal1_Rx.au8_Data[0];
gu8_MCU_MotorCoolingFlowRequest_Rx			:=	MCU_Thermal1_Rx.au8_Data[1];
gu8_MCU_ThermalIndicator_Rx					:=	MCU_Thermal1_Rx.au8_Data[2];
gq_MCU_DriveCoolingFlowRequestStatus		:=	MCU_Thermal1_Rx.au8_Data[3].0;
gq_MCU_MotorCoolingFlowRequestStatus		:=	MCU_Thermal1_Rx.au8_Data[3].1;
gq_MCU_ThermalIndicatorStatus				:=	MCU_Thermal1_Rx.au8_Data[3].2;
gu8_MCU_RollingCounter_Thermal1				:=	MCU_Thermal1_Rx.au8_Data[3] AND 2#11110000;
(*MCUPollingMCUResponse*)
gq_MCU_ResponseAcknowledgement				:=	MCU_PollingMCUResponse_Rx.au8_Data[0].0;
gu8_MCU_MCUPollResponse_Multiplex			:=	MCU_PollingMCUResponse_Rx.au8_Data[0] AND 2#01111111;
CASE gu8_MCU_MCUPollResponse_Multiplex OF
	MAXMOTORSPEED:	(*MCU MaxMotorSpeed*)
		gu16_MCU_MaxMotorSpeed_Rx			:=	USINT_TO_UINT(MCU_PollingMCUResponse_Rx.au8_Data[1]) +
												SHL(USINT_TO_UINT(MCU_PollingMCUResponse_Rx.au8_Data[2]), 8);
	MAXMOTORTORQUE:	(*MCU MaxMotorTorque*)
		gu16_MCU_MaxMotorTorque_Rx			:=	USINT_TO_UINT(MCU_PollingMCUResponse_Rx.au8_Data[1]) +
												SHL(USINT_TO_UINT(MCU_PollingMCUResponse_Rx.au8_Data[2] AND 2#01111111), 8);
	PROTOCOLVERSION:	(*MCU ProtocolVersion*)
		gu8_MCU_MajorMCUProtocol			:=	MCU_PollingMCUResponse_Rx.au8_Data[1];
		gu8_MCU_MinorMCUProtocol			:=	MCU_PollingMCUResponse_Rx.au8_Data[2];
		gu8_MCU_ExtensionMajor				:=	MCU_PollingMCUResponse_Rx.au8_Data[3];
		gu8_MCU_ExtensionMinor				:=	MCU_PollingMCUResponse_Rx.au8_Data[4];
	SWVERSION1:	(*MCU SWVersion1*)
		gu8_MCU_MajorMCUSW					:=	MCU_PollingMCUResponse_Rx.au8_Data[1];
		gu8_MCU_MinorMCUSW					:=	MCU_PollingMCUResponse_Rx.au8_Data[2];
		gu16_MCU_BranchMCUSW				:=	USINT_TO_UINT(MCU_PollingMCUResponse_Rx.au8_Data[3]) +
												SHL(USINT_TO_UINT(MCU_PollingMCUResponse_Rx.au8_Data[4]), 8);
	SWVERSION2	:(*MCU SWVersion2*)
		gu32_MCU_RevisionMCUSW				:=	USINT_TO_UDINT(MCU_PollingMCUResponse_Rx.au8_Data[1]) +
												SHL(USINT_TO_UDINT(MCU_PollingMCUResponse_Rx.au8_Data[2]), 8) +
												SHL(USINT_TO_UDINT(MCU_PollingMCUResponse_Rx.au8_Data[3]), 16) +
												SHL(USINT_TO_UDINT(MCU_PollingMCUResponse_Rx.au8_Data[4]), 24);
	TOTALMOTORROTATION:	(*MCU TotalMotorRotation*)
		gu32_MCU_TotalMotorRotation_LSB			:=	USINT_TO_UDINT(MCU_PollingMCUResponse_Rx.au8_Data[1]) +
												SHL(USINT_TO_UDINT(MCU_PollingMCUResponse_Rx.au8_Data[2]), 8) +
												SHL(USINT_TO_UDINT(MCU_PollingMCUResponse_Rx.au8_Data[3]), 16) +
												SHL(USINT_TO_UDINT(MCU_PollingMCUResponse_Rx.au8_Data[4]), 24);
		gu32_MCU_TotalMotorRotation_MSB			:=	USINT_TO_UDINT(MCU_PollingMCUResponse_Rx.au8_Data[5]) +
												SHL(USINT_TO_UDINT(MCU_PollingMCUResponse_Rx.au8_Data[6]), 8);
	TOTALMOTORROTATIONUSINTMCU:	(*MCU TotalMotorRotationUsingMCU*)
	;
ELSE
	;
END_CASE
	
(*MCUPollingVMU*)
gu8_MCU_VMUBootNumber						:=	MCU_PollingVMU_Rx.au8_Data[0];
CASE gu8_MCU_VMUBootNumber OF
	VMUBOOTNUMBER:	(*VMUBootNumber*)
		gu16_MCU_BootNumber						:=	USINT_TO_UINT(MCU_PollingVMU_Rx.au8_Data[1]) +
													SHL(USINT_TO_UINT(MCU_PollingVMU_Rx.au8_Data[2]), 8);
ELSE
	;
END_CASE
	
MCU_CommandResponse1_Rx_Timer(IN := NOT(MCU_CommandResponse1_Rx.q_NewData), PT := T#3S);
MCU_CommandResponse2_Rx_Timer(IN := NOT(MCU_CommandResponse2_Rx.q_NewData), PT := T#3S);
MCU_EventInfo1_Rx_Timer(IN := NOT(MCU_EventInfo1_Rx.q_NewData), PT := T#3S);
MCU_Info1_Rx_Timer(IN := NOT(MCU_Info1_Rx.q_NewData), PT := T#3S);
MCU_Info2_Rx_Timer(IN := NOT(MCU_Info2_Rx.q_NewData), PT := T#3S);
MCU_Thermal1_Rx_Timer(IN := NOT(MCU_Thermal1_Rx.q_NewData), PT := T#3S);
IF (MCU_CommandResponse1_Rx_Timer.Q = TRUE AND MCU_CommandResponse2_Rx_Timer.Q = TRUE AND MCU_EventInfo1_Rx_Timer.Q = TRUE AND
	MCU_Info1_Rx_Timer.Q = TRUE AND MCU_Info2_Rx_Timer.Q = TRUE AND MCU_Thermal1_Rx_Timer.Q = TRUE) THEN
	gq_MCU_CommsLoss	:=	TRUE;
ELSE
	gq_MCU_CommsLoss	:=	FALSE;
END_IF



MCU_RxConversion();

END_PROGRAM

// Application/UserCode/MCU/MCU_RxConversion_1
PROGRAM MCU_RxConversion_1
VAR
END_VAR
VAR CONSTANT
	MAXSPEED_CF		:	USINT	:=	100;
	UINT_OFFSET_CF	:	UINT	:=	32767;
	QUARTER_CF		:	REAL	:=	0.25;
	EIGHTH_CF		:	REAL	:=	0.125;
	UINT_MAX		:	UDINT	:=	65536;
	MCU_CF			:	REAL	:=	0.78125;
	CF_2POW11		:	UINT	:=	2048;
	CF_2POW12		:	UINT	:=	4096;
	
	MAX_UDINT		:	REAL	:=	4294967296;
END_VAR



gr_MCU_MaxMotorSpeedForward		:=	UINT_TO_REAL(gu16_MCU_MaxMotorSpeedForward_Rx) * MAXSPEED_CF;
gr_MCU_MaxMotorSpeedReverse		:=	UINT_TO_REAL(gu16_MCU_MaxMotorSpeedReverse_Rx) * MAXSPEED_CF;
gr_MCU_MotorSpeed				:=	UINT_TO_REAL(gu16_MCU_MotorSpeed_Rx) - UINT_OFFSET_CF;
gr_MCU_MotorAngle				:=	UINT_TO_REAL(gu16_MCU_MotorAngle_Rx) / UDINT_TO_REAL(UINT_MAX);
gr_MCU_AuxiliaryVoltage			:=	USINT_TO_REAL(gu8_MCU_AuxiliaryVoltage_Rx) * QUARTER_CF;
gr_MCU_HighPowerCurrent			:=	UINT_TO_REAL(gu16_MCU_HighPowerCurrent_Rx) * QUARTER_CF - CF_2POW11;
gr_MCU_MotorTorqueEstimated		:=	UINT_TO_REAL(gu16_MCU_MotorTorqueEstimated_Rx) * EIGHTH_CF - CF_2POW12;
gr_MCU_TractionTorqueAvailable	:=	UINT_TO_REAL(gu16_MCU_TractionTorqueAvailable_Rx) * EIGHTH_CF;
gr_MCU_RegenTorqueAvailable		:=	UINT_TO_REAL(gu16_MCU_RegenTorqueAvailable_Rx) * EIGHTH_CF;
gr_MCU_DriveCoolingFlowRequest	:=	USINT_TO_REAL(gu8_MCU_DriveCoolingFlowRequest_Rx) * MCU_CF;
gr_MCU_MotorCoolingFlowRequest	:=	USINT_TO_REAL(gu8_MCU_MotorCoolingFlowRequest_Rx) * MCU_CF;
gr_MCU_ThermalIndicator			:=	USINT_TO_REAL(gu8_MCU_ThermalIndicator_Rx) * MCU_CF;
gr_MCU_MaxMotorSpeed			:=	UINT_TO_REAL(gu16_MCU_MaxMotorSpeed_Rx) - UINT_OFFSET_CF;
gr_MCU_MaxMotorTorque			:=	UINT_TO_REAL(gu16_MCU_MaxMotorTorque_Rx) * EIGHTH_CF;

gr_MCU_TotalMotorRotation_LSB	:=	UDINT_TO_REAL(gu32_MCU_TotalMotorRotation_LSB);
gr_MCU_TotalMotorRotation_MSB	:=	UDINT_TO_REAL(gu32_MCU_TotalMotorRotation_MSB) * MAX_UDINT;
gr_MCU_TotalMotorRotation		:=	gr_MCU_TotalMotorRotation_LSB + gr_MCU_TotalMotorRotation_MSB;

END_PROGRAM

// Application/UserCode/MCU/MCU_Tx_1
PROGRAM MCU_Tx_1
VAR
	ht_MCU_VMUComm1_Tx				:	EPEC_CANVXD.Msg;
	ht_MCU_VMUComm2_Tx				:	EPEC_CANVXD.Msg;
	ht_MCU_VMUCommSafety_Tx			:	EPEC_CANVXD.Msg;
	ht_MCU_VMUPollMCU_Tx			:	EPEC_CANVXD.Msg;
	ht_MCU_VMUPollVMUResponse_Tx	:	EPEC_CANVXD.Msg;
	ht_MCU_VMUSelectProtocolVer_Tx	:	EPEC_CANVXD.Msg;
	
	(*Transmit Bytes*)
	hu8_VMUComm1_Byte1				:	USINT;
	hu8_VMUComm1_Byte5				:	USINT;
	hu8_VMUComm1_Byte7				:	USINT;
	
	hu8_VMUComm2_Byte0				:	USINT;
	
	hu8_VMUCommSafety				:	USINT;
	
	hu8_VMUPollMCU_Byte1			:	USINT;
	hu8_VMUPollMCU_Byte2			:	USINT;
	hu8_VMUPollMCU_Byte3			:	USINT;
	hu8_VMUPollMCU_Byte4			:	USINT;
	hu8_VMUPollMCU_Byte5			:	USINT;
	hu8_VMUPollMCU_Byte6			:	USINT;
	hu8_VMUPollMCU_Byte7			:	USINT;
	
	hu8_VMUPollVMUResp_Byte0		:	USINT;
	hu8_VMUPollVMUResp_Byte1		:	USINT;
	hu8_VMUPollVMUResp_Byte2		:	USINT;
	
	(*Transmit Timers*)
	hton_PeriodicSend_Timer			:	TON;
	hton_InitialisationSend_Timer	:	TON;
	
	
END_VAR


MCU_TxConversion();
(*Transmit bytes populating data*)
hu8_VMUComm1_Byte1			:=	(UINT_TO_USINT(SHR(gu16_MCU_MaxChargeCurrent, 8)) AND 2#00001111) +
								(SHL(gu8_MCU_OperationRequest, 5) AND 2#11100000);
hu8_VMUComm1_Byte5			:=	(UINT_TO_USINT(SHR(gu16_MCU_MaxBatteryVoltage, 8)) AND 2#00001111) +
								SHL(BOOL_TO_USINT(gq_MCU_MaxDiscahrgeCurrentStatus), 4) +
								SHL(BOOL_TO_USINT(gq_MCU_MaxBatteryVoltageStatus), 5) +
								SHL(BOOL_TO_USINT(gq_MCU_MinBatteryVoltageStatus), 6) +
								SHL(BOOL_TO_USINT(gq_MCU_MaxChargeCurrentStatus), 7);
hu8_VMUComm1_Byte7			:=	(UINT_TO_USINT(SHR(gu16_MCU_MinBatteryVoltage, 8)) AND 2#00001111) +
								(SHL(gu8_MCU_RollingCounter_VMUComm1, 4) AND 2#11110000);

hu8_VMUComm2_Byte0			:=	(gu8_MCU_OperationalMode_Tx AND 2#00000111) +
								(SHL(gu8_MCU_CommandMode, 3) AND 2#00011000) +
								SHL(BOOL_TO_USINT(gq_MCU_SpeedCommandStatus), 5) +
								SHL(BOOL_TO_USINT(gq_MCU_TorqueCommandStatus), 6);

hu8_VMUCommSafety			:=	(gu8_MCU_ReferenceCommandMode AND 2#00000011) +
								(SHL(gu8_MCU_RollingCounter_VMUCommSafety, 4) AND 2#11110000);

CASE gu8_MCU_VMUPollMCU_Multiplex OF
	MAXMOTORSPEED:								
		hu8_VMUPollMCU_Byte1		:=	UINT_TO_USINT(gu16_MCU_MaxMotorSpeed_Tx);
		hu8_VMUPollMCU_Byte2		:=	UINT_TO_USINT(SHR(gu16_MCU_MaxMotorSpeed_Tx, 8));
		hu8_VMUPollMCU_Byte3		:=	0;
		hu8_VMUPollMCU_Byte4		:=	0;
		hu8_VMUPollMCU_Byte5		:=	0;
		hu8_VMUPollMCU_Byte6		:=	0;
		hu8_VMUPollMCU_Byte7		:=	0;
	MAXMOTORTORQUE:								
		hu8_VMUPollMCU_Byte1		:=	UINT_TO_USINT(gu16_MCU_MaxMotorTorque_Tx);
		hu8_VMUPollMCU_Byte2		:=	UINT_TO_USINT(SHR(gu16_MCU_MaxMotorTorque_Tx, 8));
		hu8_VMUPollMCU_Byte3		:=	0;
		hu8_VMUPollMCU_Byte4		:=	0;
		hu8_VMUPollMCU_Byte5		:=	0;
		hu8_VMUPollMCU_Byte6		:=	0;
		hu8_VMUPollMCU_Byte7		:=	0;
	PROTOCOLVERSION:								
		hu8_VMUPollMCU_Byte1		:=	gu8_MCU_MajorMCUProtocol_Tx;
		hu8_VMUPollMCU_Byte2		:=	gu8_MCU_MinorMCUProtocol_Tx;
		hu8_VMUPollMCU_Byte3		:=	0;
		hu8_VMUPollMCU_Byte4		:=	0;
		hu8_VMUPollMCU_Byte5		:=	0;
		hu8_VMUPollMCU_Byte6		:=	0;
		hu8_VMUPollMCU_Byte7		:=	0;
	SWVERSION1:								
		hu8_VMUPollMCU_Byte1		:=	gu8_MCU_MajorMCUSW_Tx;
		hu8_VMUPollMCU_Byte2		:=	gu8_MCU_MinorMCUSW_Tx;
		hu8_VMUPollMCU_Byte3		:=	UINT_TO_USINT(gu16_MCU_BranchMCUSW_Tx);
		hu8_VMUPollMCU_Byte4		:=	UINT_TO_USINT(SHR(gu16_MCU_BranchMCUSW_Tx, 8));
		hu8_VMUPollMCU_Byte5		:=	0;
		hu8_VMUPollMCU_Byte6		:=	0;
		hu8_VMUPollMCU_Byte7		:=	0;
	SWVERSION2:								
		hu8_VMUPollMCU_Byte1		:=	UDINT_TO_USINT(gu32_MCU_RevisionMCUSW_Tx);
		hu8_VMUPollMCU_Byte2		:=	UDINT_TO_USINT(SHR(gu32_MCU_RevisionMCUSW_Tx, 8));
		hu8_VMUPollMCU_Byte3		:=	UDINT_TO_USINT(SHR(gu32_MCU_RevisionMCUSW_Tx, 16));
		hu8_VMUPollMCU_Byte4		:=	UDINT_TO_USINT(SHR(gu32_MCU_RevisionMCUSW_Tx, 24));
		hu8_VMUPollMCU_Byte5		:=	0;
		hu8_VMUPollMCU_Byte6		:=	0;
		hu8_VMUPollMCU_Byte7		:=	0;
	TOTALMOTORROTATION:								
		hu8_VMUPollMCU_Byte1		:=	(*UDINT_TO_USINT(gu32_MCU_TotalMotorRotation_LSB_Tx)*)0;
		hu8_VMUPollMCU_Byte2		:=	(*UDINT_TO_USINT(SHR(gu32_MCU_TotalMotorRotation_LSB_Tx, 8))*)0;
		hu8_VMUPollMCU_Byte3		:=	(*UDINT_TO_USINT(SHR(gu32_MCU_TotalMotorRotation_LSB_Tx, 16))*)0;
		hu8_VMUPollMCU_Byte4		:=	(*UDINT_TO_USINT(SHR(gu32_MCU_TotalMotorRotation_LSB_Tx, 24))*)0;
		hu8_VMUPollMCU_Byte5		:=	(*UDINT_TO_USINT(gu32_MCU_TotalMotorRotation_MSB_Tx)*)0;
		hu8_VMUPollMCU_Byte6		:=	(*UDINT_TO_USINT(SHR(gu32_MCU_TotalMotorRotation_MSB_Tx, 8))*)0;
		hu8_VMUPollMCU_Byte7		:=	0;
	TOTALMOTORROTATIONUSINTMCU:								
		hu8_VMUPollMCU_Byte1		:=	0;
		hu8_VMUPollMCU_Byte2		:=	0;
		hu8_VMUPollMCU_Byte3		:=	0;
		hu8_VMUPollMCU_Byte4		:=	0;
		hu8_VMUPollMCU_Byte5		:=	0;
		hu8_VMUPollMCU_Byte6		:=	0;
		hu8_VMUPollMCU_Byte7		:=	0;
END_CASE

hu8_VMUPollVMUResp_Byte0	:=		(gu8_MCU_PollVMUResponse_Multiplex AND 2#01111111) +
									SHL(BOOL_TO_USINT(gq_MCU_PollVMUResponse_Acknowledgement), 7);
CASE gu8_MCU_PollVMUResponse_Multiplex OF
	VMUBOOTNUMBER:
		hu8_VMUPollVMUResp_Byte1	:=	UINT_TO_USINT(gu16_MCU_BootNumber);
		hu8_VMUPollVMUResp_Byte2	:=	UINT_TO_USINT(SHR(gu16_MCU_BootNumber, 8));
END_CASE
								
								
ht_MCU_VMUComm1_Tx.ID		:=	16#040;
ht_MCU_VMUComm1_Tx.Data[0]	:=	UINT_TO_USINT(gu16_MCU_MaxChargeCurrent);
ht_MCU_VMUComm1_Tx.Data[1]	:=	hu8_VMUComm1_Byte1;
ht_MCU_VMUComm1_Tx.Data[2]	:=	UINT_TO_USINT(gu16_MCU_MaxDischargeCurrent);
ht_MCU_VMUComm1_Tx.Data[3]	:=	UINT_TO_USINT(SHR(gu16_MCU_MaxDischargeCurrent, 8)) AND 2#00001111;
ht_MCU_VMUComm1_Tx.Data[4]	:=	UINT_TO_USINT(gu16_MCU_MaxBatteryVoltage);
ht_MCU_VMUComm1_Tx.Data[5]	:=	hu8_VMUComm1_Byte5;
ht_MCU_VMUComm1_Tx.Data[6]	:=	UINT_TO_USINT(gu16_MCU_MinBatteryVoltage);
ht_MCU_VMUComm1_Tx.Data[7]	:=	hu8_VMUComm1_Byte7;
ht_MCU_VMUComm1_Tx.Len		:=	8;

ht_MCU_VMUComm2_Tx.ID		:=	16#041;
ht_MCU_VMUComm2_Tx.Data[0]	:=	hu8_VMUComm2_Byte0;
ht_MCU_VMUComm2_Tx.Data[1]	:=	UINT_TO_USINT(gu16_MCU_TorqueCommand_Tx);
ht_MCU_VMUComm2_Tx.Data[2]	:=	UINT_TO_USINT(SHR(gu16_MCU_TorqueCommand_Tx, 8));
ht_MCU_VMUComm2_Tx.Data[3]	:=	UINT_TO_USINT(gu16_MCU_SpeedCommand_Tx);
ht_MCU_VMUComm2_Tx.Data[4]	:=	UINT_TO_USINT(SHR(gu16_MCU_SpeedCommand_Tx, 8));
ht_MCU_VMUComm2_Tx.Data[5]	:=	SHL(gu8_MCU_RollingCounter_VMUComm2, 4);
ht_MCU_VMUComm2_Tx.Data[6]	:=	0;
ht_MCU_VMUComm2_Tx.Data[7]	:=	0;
ht_MCU_VMUComm2_Tx.Len		:=	6;

ht_MCU_VMUCommSafety_Tx.ID		:=	16#042;
ht_MCU_VMUCommSafety_Tx.Data[0]	:=	UINT_TO_USINT(gu16_MCU_ReferenceTorqueCommand_Tx);
ht_MCU_VMUCommSafety_Tx.Data[1]	:=	UINT_TO_USINT(SHR(gu16_MCU_ReferenceTorqueCommand_Tx, 8));
ht_MCU_VMUCommSafety_Tx.Data[2]	:=	UINT_TO_USINT(gu16_MCU_ReferenceSpeedCommand_Tx);
ht_MCU_VMUCommSafety_Tx.Data[3]	:=	UINT_TO_USINT(SHR(gu16_MCU_ReferenceSpeedCommand_Tx, 8));
ht_MCU_VMUCommSafety_Tx.Data[4]	:=	hu8_VMUCommSafety;
ht_MCU_VMUCommSafety_Tx.Data[5]	:=	0;
ht_MCU_VMUCommSafety_Tx.Data[6]	:=	0;
ht_MCU_VMUCommSafety_Tx.Data[7]	:=	0;
ht_MCU_VMUCommSafety_Tx.Len		:=	5;

ht_MCU_VMUPollMCU_Tx.ID		:=	16#447;
ht_MCU_VMUPollMCU_Tx.Data[0]	:=	gu8_MCU_VMUPollMCU_Multiplex AND 2#01111111;
ht_MCU_VMUPollMCU_Tx.Data[1]	:=	hu8_VMUPollMCU_Byte1;
ht_MCU_VMUPollMCU_Tx.Data[2]	:=	hu8_VMUPollMCU_Byte2;
ht_MCU_VMUPollMCU_Tx.Data[3]	:=	hu8_VMUPollMCU_Byte3;
ht_MCU_VMUPollMCU_Tx.Data[4]	:=	hu8_VMUPollMCU_Byte4;
ht_MCU_VMUPollMCU_Tx.Data[5]	:=	hu8_VMUPollMCU_Byte5;
ht_MCU_VMUPollMCU_Tx.Data[6]	:=	hu8_VMUPollMCU_Byte6;
ht_MCU_VMUPollMCU_Tx.Data[7]	:=	hu8_VMUPollMCU_Byte7;
ht_MCU_VMUPollMCU_Tx.Len		:=	8;

ht_MCU_VMUPollVMUResponse_Tx.ID		:=	16#446;
ht_MCU_VMUPollVMUResponse_Tx.Data[0]	:=	hu8_VMUPollVMUResp_Byte0;
ht_MCU_VMUPollVMUResponse_Tx.Data[1]	:=	hu8_VMUPollVMUResp_Byte1;
ht_MCU_VMUPollVMUResponse_Tx.Data[2]	:=	hu8_VMUPollVMUResp_Byte2;
ht_MCU_VMUPollVMUResponse_Tx.Data[3]	:=	0;
ht_MCU_VMUPollVMUResponse_Tx.Data[4]	:=	0;
ht_MCU_VMUPollVMUResponse_Tx.Data[5]	:=	0;
ht_MCU_VMUPollVMUResponse_Tx.Data[6]	:=	0;
ht_MCU_VMUPollVMUResponse_Tx.Data[7]	:=	0;
ht_MCU_VMUPollVMUResponse_Tx.Len		:=	8;

ht_MCU_VMUSelectProtocolVer_Tx.ID		:=	16#444;
ht_MCU_VMUSelectProtocolVer_Tx.Data[0]	:=	gu8_MCU_SelectMajorMCUProtocol_Tx;
ht_MCU_VMUSelectProtocolVer_Tx.Data[1]	:=	gu8_MCU_SelectMinorMCUProtocol_Tx;
ht_MCU_VMUSelectProtocolVer_Tx.Data[2]	:=	0;
ht_MCU_VMUSelectProtocolVer_Tx.Data[3]	:=	0;
ht_MCU_VMUSelectProtocolVer_Tx.Data[4]	:=	0;
ht_MCU_VMUSelectProtocolVer_Tx.Data[5]	:=	0;
ht_MCU_VMUSelectProtocolVer_Tx.Data[6]	:=	0;
ht_MCU_VMUSelectProtocolVer_Tx.Data[7]	:=	0;
ht_MCU_VMUSelectProtocolVer_Tx.Len		:=	2;


IF (gu8_MCU_MajorMCUProtocol = 0(* AND gq_InitialProtocolGrab = FALSE*)) THEN
	hton_InitialisationSend_Timer(IN := NOT(hton_InitialisationSend_Timer.Q), PT := T#10MS);
	IF (hton_InitialisationSend_Timer.Q = TRUE) THEN
		G_CAN1_Channel.SendMessage(i_pMSG:=ADR(ht_MCU_VMUSelectProtocolVer_Tx));
	END_IF
ELSIF (gu8_MCU_MajorMCUProtocol <> 0) THEN
	(*hton_PeriodicSend_Timer(IN := TRUE, PT := T#10MS);*)
	IF (hton_PeriodicSend_Timer.Q = (*TRUE*)FALSE) THEN
		G_CAN1_Channel.SendMessage(i_pMSG:=ADR(ht_MCU_VMUComm1_Tx));
		G_CAN1_Channel.SendMessage(i_pMSG:=ADR(ht_MCU_VMUComm2_Tx));
		G_CAN1_Channel.SendMessage(i_pMSG:=ADR(ht_MCU_VMUCommSafety_Tx));
		IF (gu8_MCU_VMUPollMCU_Multiplex >= 0 AND gu8_MCU_VMUPollMCU_Multiplex < 8) THEN
			G_CAN1_Channel.SendMessage(i_pMSG:=ADR(ht_MCU_VMUPollMCU_Tx));
		END_IF
		gu8_MCU_RollingCounter_VMUComm1			:=	gu8_MCU_RollingCounter_VMUComm1 + 1;
		gu8_MCU_RollingCounter_VMUComm2			:=	gu8_MCU_RollingCounter_VMUComm2 + 1;
		gu8_MCU_RollingCounter_VMUCommSafety	:=	gu8_MCU_RollingCounter_VMUCommSafety + 1;
		IF (gu8_MCU_RollingCounter_VMUComm1 > 15) THEN
			gu8_MCU_RollingCounter_VMUComm1	:=	0;
		END_IF
		IF (gu8_MCU_RollingCounter_VMUComm2 > 15) THEN
			gu8_MCU_RollingCounter_VMUComm2	:=	0;
		END_IF
		IF (gu8_MCU_RollingCounter_VMUCommSafety > 15) THEN
			gu8_MCU_RollingCounter_VMUCommSafety	:=	0;
		END_IF
		(*Update the last command value sent*)
		gr_MCU_PreviousTorqueCommand		:=	gr_MCU_TorqueCommand_Limited;
		hton_PeriodicSend_Timer(IN := FALSE, PT := T#0MS);
	END_IF
	gq_InitialProtocolGrab	:=	TRUE;
END_IF

END_PROGRAM

// Application/UserCode/MCU/MCU_TxConversion_1
PROGRAM MCU_TxConversion_1
VAR
	hr_MCU_LowerLimitTorqueCommand	:	REAL;
	hr_MCU_UpperLimitTorqueCommand	:	REAL;
	LowPassFilter	:	OSCAT_BASIC.FT_PT1;
	TimeConstant	:	REAL	:=	1000;
END_VAR
VAR RETAIN
	hr_INCREASETORQUERAMP	:	REAL	:=	3500; (*Nm/s*)
	hr_DECREASETORQUERAMP	:	REAL	:=	7000; (*Nm/s*)
END_VAR


(*10ms *)
(*
hr_MCU_LowerLimitTorqueCommand		:=	gr_MCU_PreviousTorqueCommand - (hr_DECREASETORQUERAMP / 100);
hr_MCU_UpperLimitTorqueCommand		:=	gr_MCU_PreviousTorqueCommand + (hr_INCREASETORQUERAMP / 100);
gr_MCU_TorqueCommand_Limited		:=	LIMIT(hr_MCU_LowerLimitTorqueCommand, gr_MCU_TorqueCommand_PreCF_Limited, hr_MCU_UpperLimitTorqueCommand);
*)
LowPassFilter(in := gr_MCU_TorqueCommand_PreCF_Limited, T := REAL_TO_TIME(TimeConstant), K := 1, out => gr_MCU_TorqueCommand_Limited);


gu16_MCU_TorqueCommand_Tx			:=	REAL_TO_UINT((gr_MCU_TorqueCommand_Limited + 4096) / 0.125);
gu16_MCU_SpeedCommand_Tx			:=	REAL_TO_UINT(gr_MCU_SpeedCommand_PreCF) + 32767;
gu16_MCU_ReferenceTorqueCommand_Tx	:=	REAL_TO_UINT((gr_MCU_ReferenceTorqueCommand_PreCF + 4096) / 0.125);
gu16_MCU_ReferenceSpeedCommand_Tx	:=	REAL_TO_UINT(gr_MCU_ReferenceSpeedCommand_PreCF) + 32767;
gu16_MCU_MaxMotorSpeed_Tx			:=	REAL_TO_UINT(gr_MCU_MaxMotorSpeed_PreCF + 32767);
gu16_MCU_MaxMotorTorque_Tx			:=	REAL_TO_UINT(4000 / 0.125); (*Not currently sent as the max torque is gained from the MCU*)

gu8_MCU_SelectMajorMCUProtocol_Tx	:=	4;
gu8_MCU_SelectMinorMCUProtocol_Tx	:=	0;

END_PROGRAM

// Application/UserCode/Sevcon_Compressor/Sevcon2_Control_1
PROGRAM Sevcon2_Control_1
VAR
	hton_WindUpTorque_Timer	:	TON;
	hton_AirPressureExceeded_Timer	:	TON;
	htof_AirpressureRelief_Timer	:	TOF;
	hq_AirCompressorEnable	:	BOOL;
	hton_AirPressureDelayTimer	:	TON;
	
	hq_AirReliefValveOff : BOOL;
	
	
	hton_Compressor_Oil_Switch: TON;
	Low_Oil: BOOL;
	NO_OIL: BOOL;
	Oil_Temp_Setpoint: BYTE := 30;
	Oil_Level_Warning: BOOL;
	Compressor_Temp_Warning: BOOL;
	Comp_Motor_Temp_SP_Warning: INT := 100; //LM change from 55
	Comp_Motor_Temp_SP_Fault: INT := 120;  //LM change from 65
	Compressor_Temp_Fault: BOOL;
	Air_Temp_SP_Warning: INT := 100;
	Air_Temp_SP_Fault: INT := 120;
	Air_Temp_Warning: BOOL;
	Air_Temp_Fault: BOOL;
	BlowOffTime: TIME := T#1S;
	AirSuspensionPressure: REAL := 14.9;
	APRTimerET: TIME := t#0.5s;
	AirPressureReliefTime: TIME := t#1s;
	hton_Compressor_Run_Timer: TON;
	CRT_Trigger: BOOL;
	CRT_Time: TIME := t#60s;
	Run_on_Brake_Pressure: REAL := 9.5;
	CRT_Timer: TON;
	PVCT: TON;
	PVCT_Time: TIME := T#60s;
END_VAR
VAR CONSTANT
	(*Statuswords*)
	NOTREADY_STAT				:	USINT	:=	1;
	SHUTDOWN_STAT				:	USINT	:=	2;
	PRECHARGE_STAT				:	USINT	:=	4;
	ENERGISED_STAT				:	USINT	:=	7;
	ENABLED_STAT				:	USINT	:=	8;
	FAULTREACTIONACTIVE_STAT	:	USINT	:=	11;
	FAULTOFF_STAT				:	USINT	:=	13;
	ACTIVESHORT_STAT			:	USINT	:=	14;
	(*Commandwords*)
	NOCOMMAND_COMM		:	USINT	:=	0;
	ENERGISE_COMM		:	USINT	:=	3;
	ENABLED_COMM		:	USINT	:=	5;
	SHUTDOWN_COMM		:	USINT	:=	6;
	FAULTRESET_COMM		:	USINT	:=	9;
	ACTIVESHORT_COMM	:	USINT	:=	10;
	
	(*LOWAIRPRESSURE		:	REAL	:=	7.2; (*Need to define what the low air pressure value that is reported is*)
	HIGHAIRPRESSURE		:	REAL	:=	10;
	LOWAIRPRESSURE_BOB		:	REAL	:=	10; (*Need to define what the low air pressure value that is reported is*)
	HIGHAIRPRESSURE_BOB		:	REAL	:=	12.2(*Glider*) (*12.3 for Bob*);*)
	
	
	TORQUE_RQ			:	USINT	:=	200;
	REVERSE_SPD_LIMIT	:	INT		:=	-500;
	MAX_DISCHARGE		:	USINT	:=	50;
	MAX_CHARGE			:	SINT	:=	-50;
	TRACTION_LIMIT		:	USINT	:=	100;
END_VAR


(**)
(*Check for Comms fault*)
IF (gu8_SystemState = DRIVE_SYS AND DOS_q_BatteryDischargeMain_DO = TRUE) THEN
	IF (gu8_Sevcon2_InverterStatus = FAULTOFF_STAT OR gu8_Sevcon2_InverterStatus = ACTIVESHORT_STAT) THEN
		gu16_Sevcon2_Controlword	:=	FAULTRESET_COMM;
	ELSIF (gu8_Sevcon2_InverterStatus = NOTREADY_STAT OR gu8_Sevcon2_InverterStatus = SHUTDOWN_STAT) THEN
		gu16_Sevcon2_Controlword	:=	ENERGISE_COMM;
	ELSIF (gu8_Sevcon2_InverterStatus = PRECHARGE_STAT) THEN
		gu16_Sevcon2_Controlword	:=	ENERGISE_COMM;
	ELSIF (gu8_Sevcon2_InverterStatus = ENERGISED_STAT) THEN
		gu16_Sevcon2_Controlword	:=	ENABLED_COMM;
	ELSIF (gu8_Sevcon2_InverterStatus = ENABLED_STAT) THEN
		gu16_Sevcon2_Controlword	:=	ENABLED_COMM; (*Need a way to switch off*)
	ELSE
		gu16_Sevcon2_Controlword	:=	NOCOMMAND_COMM;
	END_IF
ELSE
	gu16_Sevcon2_Controlword	:=	SHUTDOWN_COMM;
END_IF

CRT_Timer (IN:= NOT hq_AirCompressorEnable, PT := CRT_Time); //Active when compressor hasnt run
hton_AirPressureDelayTimer(IN := TRUE, PT := T#2000MS);
PVCT (IN :=  hq_AirCompressorEnable, PT := PVCT_Time); // Compressor run-on timer

IF (hton_AirPressureDelayTimer.Q = TRUE) THEN
	IF (gq_APU_Installed = FALSE) THEN
		IF 	//(gr_J1939_AirSuspensionSupplyPress > gr_HighAirPressure_CutOff OR
			(gr_J1939_ServiceBrakeAirPressCircuit1 > gr_HighAirPressure_CutOff OR
			gr_J1939_ServiceBrakeAirPressCircuit2 > gr_HighAirPressure_CutOff) THEN
			hton_AirPressureExceeded_Timer(IN := TRUE, PT := BlowOffTime);
		ELSE
			hton_AirPressureExceeded_Timer(IN := FALSE, PT := T#1S); //changed from 0 to 2s to increase hysteresis
		END_IF
		IF (gu8_SystemState = DRIVE_SYS AND DOS_q_BatteryDischargeMain_DO = TRUE AND
			NO_OIL = FALSE AND Compressor_Temp_Fault = FALSE) (*AND gq_Bob_AirCompressorStatus_CAN = TRUE)*) THEN
			IF  (gr_VehicleSpeed_kmph > 5 AND (gr_J1939_ServiceBrakeAirPressCircuit1 < Run_on_Brake_Pressure)) OR // added to increase duty cycle
				
				//(PVCT.Q = FALSE AND CRT_Timer.Q = TRUE AND gr_VehicleSpeed_kmph > 2) OR // runs compressor for a time period
				
				((gr_J1939_AirSuspensionSupplyPress < gr_LowAirPressure_Intro OR
				gr_J1939_ServiceBrakeAirPressCircuit1 < gr_LowAirPressure_Intro OR
				gr_J1939_ServiceBrakeAirPressCircuit2 < gr_LowAirPressure_Intro)) THEN
					gu16_Sevcon2_SpeedLimitForward	:=	2600; (*Controlling the speed through the limits*)
					hq_AirCompressorEnable	:=	TRUE;
			ELSIF ((hton_AirPressureExceeded_Timer.Q = TRUE) OR (gr_VehicleSpeed_kmph > 5 AND (gr_J1939_ServiceBrakeAirPressCircuit1 > Run_on_Brake_Pressure))) THEN
				//(PVCT.Q = TRUE AND CRT_Timer.Q = FALSE AND gr_VehicleSpeed_kmph < 2) THEN // added to increase duty cycle
				gu16_Sevcon2_SpeedLimitForward	:=	0;
				hq_AirCompressorEnable	:=	FALSE;
			END_IF
		ELSE
			gu16_Sevcon2_SpeedLimitForward	:=	0;
			hq_AirCompressorEnable	:=	FALSE;
		END_IF
	
	(*For Bob possibly use
	(*gq_Bob_AirCompressorStatus_CAN = FALSE AND hq_AirReliefValveOff = TRUE)*)
	See below for how it was implemented*)
		
	(*This is needed for when the compressor is being controlled by the APU not yet*)
	ELSE
		(*IF (gr_J1939_AirSuspensionSupplyPress > HIGHAIRPRESSURE_BOB AND
			(gr_J1939_ServiceBrakeAirPressCircuit1 > HIGHAIRPRESSURE_BOB AND
			gr_J1939_ServiceBrakeAirPressCircuit2 > HIGHAIRPRESSURE_BOB))				
			(*gq_Bob_AirCompressorStatus_CAN = FALSE AND hq_AirReliefValveOff = TRUE)*) THEN
			hton_AirPressureExceeded_Timer(IN := TRUE, PT := T#1000MS);
		ELSE
			hton_AirPressureExceeded_Timer(IN := FALSE, PT := T#0MS);
		END_IF*)
		IF (gu8_SystemState = DRIVE_SYS AND DOS_q_BatteryDischargeMain_DO = TRUE AND
			NO_OIL = FALSE AND Compressor_Temp_Fault = FALSE AND gq_Bob_AirCompressorStatus_CAN = TRUE) THEN
			IF (gq_Merc_AirComp_Rq = TRUE) OR (htof_AirpressureRelief_Timer.ET > APRTimerET) THEN
					gu16_Sevcon2_SpeedLimitForward	:=	2600; (*Controlling the speed through the limits*)
					hq_AirCompressorEnable	:=	TRUE;
			ELSE(*ELSIF (hton_AirPressureExceeded_Timer.Q = TRUE) THEN*)
				gu16_Sevcon2_SpeedLimitForward	:=	0;
				hq_AirCompressorEnable	:=	FALSE;
			END_IF
		ELSE
			gu16_Sevcon2_SpeedLimitForward	:=	0;
			hq_AirCompressorEnable	:=	FALSE;
		END_IF
		(*hq_AirReliefValveOff := gq_Bob_AirCompressorStatus_CAN;*)
	END_IF
END_IF
(*gq_Merc_AirComp_Enabled	:=	hq_AirCompressorEnable;*)


htof_AirpressureRelief_Timer(IN := gq_Merc_AirComp_Rq, PT := AirPressureReliefTime);
IF htof_AirpressureRelief_Timer.Q THEN
	hq_AirCompressorEnable	:=	TRUE;
	(*(hq_AirCompressorEnable = TRUE AND gs16_Sevcon2_SpeedMeasured < 1000 )) THEN*)
	gu16_Sevcon2_SpeedLimitForward	:=	2600; (*Controlling the speed through the limits*)
	hq_AirCompressorEnable	:=	TRUE;
ELSE
		;
END_IF


(*All these are constants to be sent out to the Sevcon unit and do not need changing during operation*)
IF (gu8_Sevcon2_InverterStatus = ENABLED_STAT) THEN
	hton_WindUpTorque_Timer(IN := TRUE, PT := T#5000MS);
	gr_Sevcon2_TorqueRq						:=	TORQUE_RQ * (TIME_TO_REAL(hton_WindUpTorque_Timer.ET) / 5000);
ELSE
	hton_WindUpTorque_Timer(IN := FALSE, PT := T#0MS);
	gr_Sevcon2_TorqueRq						:=	0;
END_IF
	
gr_Sevcon2_DCLink_VoltageTarget			:=	0; (*Not needed as not being used as a generator*)
gs16_Sevcon2_SpeedLimitReverse			:=	REVERSE_SPD_LIMIT;
gu16_Sevcon2_DCLink_ImaxDischarge		:=	MAX_DISCHARGE;
gs16_Sevcon2_DCLink_ImaxRecharge		:=	MAX_CHARGE;
gr_Sevcon2_TorqueTractionLimit			:=	TRACTION_LIMIT;
gr_Sevcon2_TorqueRegenLimit				:=	0;

gu8_Sevcon2_CSCommand1					:=	0;
gu8_Sevcon2_CSCommand2					:=	0;
gu8_Sevcon2_CSCurrentLimits				:=	0;
(*Counters to run every cycle and increment so the Sevcons know the VMU is still running*)
IF (gu8_Sevcon2_SEQCommand1 < 255) THEN
	gu8_Sevcon2_SEQCommand1			:=	gu8_Sevcon2_SEQCommand1 + 1;
ELSE
	gu8_Sevcon2_SEQCommand1			:=	0;
END_IF
IF (gu8_Sevcon2_SEQCommand2 < 255) THEN
	gu8_Sevcon2_SEQCommand2			:=	gu8_Sevcon2_SEQCommand2 + 1;
ELSE
	gu8_Sevcon2_SEQCommand2			:=	0;
END_IF
IF (gu8_Sevcon2_SEQCurrentLimits < 255) THEN
	gu8_Sevcon2_SEQCurrentLimits	:=	gu8_Sevcon2_SEQCurrentLimits + 1;
ELSE
	gu8_Sevcon2_SEQCurrentLimits	:=	0;
END_IF
(**************************************************************)
hton_Compressor_Oil_Switch(IN:= Low_Oil, PT:= T#2M);
IF Sevcon2_Rx.Compressor_Oil_Switch < 1 (*Rimmed AND gs16_Sevcon2_MotorTemp < Oil_Temp_Setpoint *) AND  gs16_Sevcon2_SpeedMeasured <2000 THEN
	Low_Oil := FALSE; (*changed due to poor switching*)
ELSE
	Low_Oil := FALSE;
END_IF

IF hton_Compressor_Oil_Switch.Q THEN
	NO_OIL := FALSE;
ELSE
	NO_OIL := FALSE;
END_IF

IF hton_Compressor_Oil_Switch.ET > T#30S THEN
	Oil_Level_Warning := TRUE;
ELSE
	Oil_Level_Warning := FALSE;
END_IF

IF gs16_Sevcon2_MotorTemp > Comp_Motor_Temp_SP_Warning THEN
	Compressor_Temp_Warning	:= TRUE;
ELSE
	Compressor_Temp_Warning	:= FALSE;
END_IF

IF	gs16_Sevcon2_MotorTemp > Comp_Motor_Temp_SP_Fault THEN
	Compressor_Temp_Fault := TRUE;
ELSE
	Compressor_Temp_fault := FALSE;
END_IF

IF	Sevcon2_Rx.Compressor_Temperature > Air_Temp_SP_Warning THEN
	Air_Temp_Warning := TRUE;
ELSE
	Air_Temp_Warning := FALSE;
END_IF

IF	Sevcon2_Rx.Compressor_Temperature > Air_Temp_SP_Fault THEN
	Air_Temp_Fault := TRUE;
ELSE
	Air_Temp_Fault := FALSE;
END_IF

END_PROGRAM

// Application/UserCode/Sevcon_Compressor/Sevcon2_Rx_1
PROGRAM Sevcon2_Rx_1
VAR
	Compressor_Oil_Rx	:	Receive_CAN2_EXD;
	Compressor_Temp_Rx	:	Receive_CAN2_STD;
	TorqueStatus1_Rx	:	Receive_CAN2_EXD;
	TorqueStatus2_Rx	:	Receive_CAN2_EXD;
	TempStatus_Rx		:	Receive_CAN2_EXD;
	FaultStatus_Rx		:	Receive_CAN2_EXD;
	EncoderStatus_Rx	:	Receive_CAN2_EXD;
	DeubgCurrents_Rx	:	Receive_CAN2_EXD;
	DebugTemps1_Rx		:	Receive_CAN2_EXD;
	DebugTemps2_Rx		:	Receive_CAN2_EXD;
	DebugPMACControl_Rx	:	Receive_CAN2_EXD;
	DebugFVControl_Rx	:	Receive_CAN2_EXD;
	
	TorqueStatus1_Rx_Timer		:	TON;
	TorqueStatus2_Rx_Timer		:	TON;
	TempStatus_Rx_Timer			:	TON;
	FaultStatus_Rx_Timer		:	TON;
	EncoderStatus_Rx_Timer		:	TON;
	DeubgCurrents_Rx_Timer		:	TON;
	DebugTemps1_Rx_Timer		:	TON;
	DebugTemps2_Rx_Timer		:	TON;
	DebugPMACControl_Rx_Timer	:	TON;
	DebugFVControl_Rx_Timer		:	TON;
	Compressor_Temperature		: 	INT;
	Compressor_Oil_Switch		:	BYTE;
	
END_VAR

Compressor_Oil_Rx(u32_COBID	:=	16#1948FF72,
				q_NewData => ,
				au8_Data => ,
				u8_Length => 			);

Compressor_Temp_Rx(u32_COBID	:=	16#443,
				q_NewData => ,
				au8_Data => ,
				u8_Length => 			);

TorqueStatus1_Rx(u32_COBID	:=	16#1918FF72,
				q_NewData => ,
				au8_Data => ,
				u8_Length => 			);

TorqueStatus2_Rx(u32_COBID	:=	16#1919FF72,
				q_NewData => ,
				au8_Data => ,
				u8_Length => 			);

TempStatus_Rx(u32_COBID	:=	16#191AFF72,
				q_NewData => ,
				au8_Data => ,
				u8_Length => 			);

FaultStatus_Rx(u32_COBID	:=	16#191BFF72,
				q_NewData => ,
				au8_Data => ,
				u8_Length => 			);

EncoderStatus_Rx(u32_COBID	:=	16#191CFF72,
				q_NewData => ,
				au8_Data => ,
				u8_Length => 			);

DeubgCurrents_Rx(u32_COBID	:=	16#1928FF72,
				q_NewData => ,
				au8_Data => ,
				u8_Length => 			);

DebugTemps1_Rx(u32_COBID	:=	16#192AFF72,
				q_NewData => ,
				au8_Data => ,
				u8_Length => 			);

DebugTemps2_Rx(u32_COBID	:=	16#192BFF72,
				q_NewData => ,
				au8_Data => ,
				u8_Length => 			);

DebugPMACControl_Rx(u32_COBID	:=	16#192CFF72,
				q_NewData => ,
				au8_Data => ,
				u8_Length => 			);

DebugFVControl_Rx(u32_COBID	:=	16#192DFF72,
				q_NewData => ,
				au8_Data => ,
				u8_Length => 			);				

Compressor_Oil_Switch					:=	BIT_TO_BYTE (Compressor_Oil_Rx.au8_Data[2].4) +
											BIT_TO_BYTE (Compressor_Oil_Rx.au8_Data[2].5);

Compressor_Temperature					:=	Compressor_Temp_Rx.au8_Data[5] +
											Compressor_Temp_Rx.au8_Data[6];
				
gs16_Sevcon2_TorqueMeasured_Rx			:=	USINT_TO_INT(TorqueStatus1_Rx.au8_Data[0]) +
											SHL(USINT_TO_INT(TorqueStatus1_Rx.au8_Data[1]), 8);
gs16_Sevcon2_SpeedMeasured				:=	USINT_TO_INT(TorqueStatus1_Rx.au8_Data[2]) +
											SHL(USINT_TO_INT(TorqueStatus1_Rx.au8_Data[3]), 8);
gs16_Sevcon2_DCLink_Current				:=	USINT_TO_INT(TorqueStatus1_Rx.au8_Data[4]) +
											SHL(USINT_TO_INT(TorqueStatus1_Rx.au8_Data[5]), 8);
gu8_Sevcon2_SEQ_Torque					:=	TorqueStatus1_Rx.au8_Data[6];
gu8_Sevcon2_CS_Torque					:=	TorqueStatus1_Rx.au8_Data[7];

gs16_Sevcon2_TorqueAvailableForward_Rx	:=	USINT_TO_INT(TorqueStatus2_Rx.au8_Data[0]) +
											SHL(USINT_TO_INT(TorqueStatus2_Rx.au8_Data[1]), 8);
gs16_Sevcon2_TorqueAvailableReverse_Rx	:=	USINT_TO_INT(TorqueStatus2_Rx.au8_Data[2]) +
											SHL(USINT_TO_INT(TorqueStatus2_Rx.au8_Data[3]), 8);
gu8_Sevcon2_InverterStatus				:=	TorqueStatus2_Rx.au8_Data[4];
gu8_Sevcon2_TorqueLimitCode				:=	TorqueStatus2_Rx.au8_Data[5];
gu8_Sevcon2_SEQ_Status					:=	TorqueStatus2_Rx.au8_Data[6];
gu8_Sevcon2_CS_Status					:=	TorqueStatus2_Rx.au8_Data[7];

gs16_Sevcon2_TempRemaining				:=	USINT_TO_INT(TempStatus_Rx.au8_Data[0]) +
											SHL(USINT_TO_INT(TempStatus_Rx.au8_Data[1]), 8);
gs16_Sevcon2_MotorTemp					:=	USINT_TO_INT(TempStatus_Rx.au8_Data[2]) +
											SHL(USINT_TO_INT(TempStatus_Rx.au8_Data[3]), 8);
gs16_Sevcon2_DCLink_Voltage_Rx			:=	USINT_TO_INT(TempStatus_Rx.au8_Data[4]) +
											SHL(USINT_TO_INT(TempStatus_Rx.au8_Data[5]), 8);
gu8_Sevcon2_SEQ_Temp					:=	TempStatus_Rx.au8_Data[6];
gu8_Sevcon2_CS_Temp						:=	TempStatus_Rx.au8_Data[7];

gs16_Sevcon2_FaultCode					:=	USINT_TO_INT(FaultStatus_Rx.au8_Data[0]) +
											SHL(USINT_TO_INT(FaultStatus_Rx.au8_Data[1]), 8);
gs32_Sevcon2_FaultData					:=	USINT_TO_DINT(FaultStatus_Rx.au8_Data[2]) +
											SHL(USINT_TO_DINT(FaultStatus_Rx.au8_Data[3]), 8) +
											SHL(USINT_TO_DINT(FaultStatus_Rx.au8_Data[4]), 16) +
											SHL(USINT_TO_DINT(FaultStatus_Rx.au8_Data[5]), 24);
gu8_Sevcon2_SEQ_Fault					:=	FaultStatus_Rx.au8_Data[6];
gu8_Sevcon2_CS_Fault					:=	FaultStatus_Rx.au8_Data[7];

gs32_Sevcon2_EncoderPosition_Rx			:=	USINT_TO_DINT(EncoderStatus_Rx.au8_Data[0]) +
											SHL(USINT_TO_DINT(EncoderStatus_Rx.au8_Data[1]), 8) +
											SHL(USINT_TO_DINT(EncoderStatus_Rx.au8_Data[2]), 16) +
											SHL(USINT_TO_DINT(EncoderStatus_Rx.au8_Data[3]), 24);

gs16_Sevcon2_Debug_Id_Act_Rx			:=	USINT_TO_INT(DeubgCurrents_Rx.au8_Data[0]) +
											SHL(USINT_TO_INT(DeubgCurrents_Rx.au8_Data[1]), 8);
gs16_Sevcon2_Debug_Iq_Act_Rx			:=	USINT_TO_INT(DeubgCurrents_Rx.au8_Data[2]) +
											SHL(USINT_TO_INT(DeubgCurrents_Rx.au8_Data[3]), 8);
gs16_Sevcon2_Debug_Id_Ref_Rx			:=	USINT_TO_INT(DeubgCurrents_Rx.au8_Data[4]) +
											SHL(USINT_TO_INT(DeubgCurrents_Rx.au8_Data[5]), 8);
gs16_Sevcon2_Debug_Iq_Ref_Rx			:=	USINT_TO_INT(DeubgCurrents_Rx.au8_Data[6]) +
											SHL(USINT_TO_INT(DeubgCurrents_Rx.au8_Data[7]), 8);

gu8_Sevcon2_Debug_Temp_Junction0		:=	DebugTemps1_Rx.au8_Data[0];
gu8_Sevcon2_Debug_Temp_Junction1		:=	DebugTemps1_Rx.au8_Data[1];
gu8_Sevcon2_Debug_Temp_Junction2		:=	DebugTemps1_Rx.au8_Data[2];
gu8_Sevcon2_Debug_Temp_Junction3		:=	DebugTemps1_Rx.au8_Data[3];
gu8_Sevcon2_Debug_Temp_Junction4		:=	DebugTemps1_Rx.au8_Data[4];
gu8_Sevcon2_Debug_Temp_Junction5		:=	DebugTemps1_Rx.au8_Data[5];
gu8_Sevcon2_Debug_Temp_MotorMeasured	:=	DebugTemps1_Rx.au8_Data[6];
gu8_Sevcon2_Debug_Temp_MotorEstimate	:=	DebugTemps1_Rx.au8_Data[7];

gu8_Sevcon2_Debug_Temp_CapEstimateFast	:=	DebugTemps2_Rx.au8_Data[0];
gu8_Sevcon2_Debug_Temp_Track			:=	DebugTemps2_Rx.au8_Data[1];
gu8_Sevcon2_Debug_Temp_CapEstimateSlow	:=	DebugTemps2_Rx.au8_Data[2];
gu8_Sevcon2_Debug_Temp_Heatsink			:=	DebugTemps2_Rx.au8_Data[3];
gu8_Sevcon2_Debug_Temp_DeltaTj			:=	DebugTemps2_Rx.au8_Data[4];
gu8_Sevcon2_Debug_Temp_Normalised		:=	DebugTemps2_Rx.au8_Data[5];
gu8_Sevcon2_Debug_Temp_Coolant			:=	DebugTemps2_Rx.au8_Data[6];
gu8_Sevcon2_Debug_Temp_Winding			:=	DebugTemps2_Rx.au8_Data[7];

